//     PlcTask Inputs/GVL_iXlinker.EtherCAT_Master_ATxxxx.Beckhoff_ATH2xxx.Beckhoff_ATH2xxxEK1122.A_0004_ATH2040_0250_0022.InfoData.State <-> InfoData/State
//   PLC/PLC Instance <-> EtherCAT Master ATxxxx/Beckhoff ATH2xxx/Beckhoff ATH2xxxEK1122/A_0005(ATH2040-0250-0023)
//     PlcTask Inputs/GVL_iXlinker.EtherCAT_Master_ATxxxx.Beckhoff_ATH2xxx.Beckhoff_ATH2xxxEK1122.A_0005_ATH2040_0250_0023.CC_Inputs.Status <-> CC Inputs/Status
//     PlcTask Inputs/GVL_iXlinker.EtherCAT_Master_ATxxxx.Beckhoff_ATH2xxx.Beckhoff_ATH2xxxEK1122.A_0005_ATH2040_0250_0023.CC_Inputs.Current_actual_value_Ch[0] <-> CC Inputs/Current actual value Ch.1
//     PlcTask Inputs/GVL_iXlinker.EtherCAT_Master_ATxxxx.Beckhoff_ATH2xxx.Beckhoff_ATH2xxxEK1122.A_0005_ATH2040_0250_0023.CC_Inputs.Current_actual_value_Ch[1] <-> CC Inputs/Current actual value Ch.2
//     PlcTask Inputs/GVL_iXlinker.EtherCAT_Master_ATxxxx.Beckhoff_ATH2xxx.Beckhoff_ATH2xxxEK1122.A_0005_ATH2040_0250_0023.CC_Inputs.Current_actual_value_Ch[2] <-> CC Inputs/Current actual value Ch.3
//     PlcTask Inputs/GVL_iXlinker.EtherCAT_Master_ATxxxx.Beckhoff_ATH2xxx.Beckhoff_ATH2xxxEK1122.A_0005_ATH2040_0250_0023.CC_Inputs.Current_actual_value_Ch[3] <-> CC Inputs/Current actual value Ch.4
//     PlcTask Inputs/GVL_iXlinker.EtherCAT_Master_ATxxxx.Beckhoff_ATH2xxx.Beckhoff_ATH2xxxEK1122.A_0005_ATH2040_0250_0023.CC_Inputs.Current_actual_value_Ch[4] <-> CC Inputs/Current actual value Ch.5
//     PlcTask Inputs/GVL_iXlinker.EtherCAT_Master_ATxxxx.Beckhoff_ATH2xxx.Beckhoff_ATH2xxxEK1122.A_0005_ATH2040_0250_0023.CC_Inputs.Current_actual_value_Ch[5] <-> CC Inputs/Current actual value Ch.6
//     PlcTask Inputs/GVL_iXlinker.EtherCAT_Master_ATxxxx.Beckhoff_ATH2xxx.Beckhoff_ATH2xxxEK1122.A_0005_ATH2040_0250_0023.CC_Inputs.Current_actual_value_Ch[6] <-> CC Inputs/Current actual value Ch.7
//     PlcTask Inputs/GVL_iXlinker.EtherCAT_Master_ATxxxx.Beckhoff_ATH2xxx.Beckhoff_ATH2xxxEK1122.A_0005_ATH2040_0250_0023.CC_Inputs.Current_actual_value_Ch[7] <-> CC Inputs/Current actual value Ch.8
//     PlcTask Inputs/GVL_iXlinker.EtherCAT_Master_ATxxxx.Beckhoff_ATH2xxx.Beckhoff_ATH2xxxEK1122.A_0005_ATH2040_0250_0023.CC_Inputs.Current_actual_value_Ch[8] <-> CC Inputs/Current actual value Ch.9
//     PlcTask Inputs/GVL_iXlinker.EtherCAT_Master_ATxxxx.Beckhoff_ATH2xxx.Beckhoff_ATH2xxxEK1122.A_0005_ATH2040_0250_0023.CC_Inputs.Current_actual_value_Ch[9] <-> CC Inputs/Current actual value Ch.10
//     PlcTask Inputs/GVL_iXlinker.EtherCAT_Master_ATxxxx.Beckhoff_ATH2xxx.Beckhoff_ATH2xxxEK1122.A_0005_ATH2040_0250_0023.CC_Inputs.Current_actual_value_Ch[10] <-> CC Inputs/Current actual value Ch.11
//     PlcTask Inputs/GVL_iXlinker.EtherCAT_Master_ATxxxx.Beckhoff_ATH2xxx.Beckhoff_ATH2xxxEK1122.A_0005_ATH2040_0250_0023.CC_Inputs.Current_actual_value_Ch[11] <-> CC Inputs/Current actual value Ch.12
//     PlcTask Inputs/GVL_iXlinker.EtherCAT_Master_ATxxxx.Beckhoff_ATH2xxx.Beckhoff_ATH2xxxEK1122.A_0005_ATH2040_0250_0023.CC_Inputs.Current_actual_value_Ch[12] <-> CC Inputs/Current actual value Ch.13
//     PlcTask Inputs/GVL_iXlinker.EtherCAT_Master_ATxxxx.Beckhoff_ATH2xxx.Beckhoff_ATH2xxxEK1122.A_0005_ATH2040_0250_0023.CC_Inputs.Current_actual_value_Ch[13] <-> CC Inputs/Current actual value Ch.14
//     PlcTask Inputs/GVL_iXlinker.EtherCAT_Master_ATxxxx.Beckhoff_ATH2xxx.Beckhoff_ATH2xxxEK1122.A_0005_ATH2040_0250_0023.CC_Inputs.Current_actual_value_Ch[14] <-> CC Inputs/Current actual value Ch.15
//     PlcTask Outputs/GVL_iXlinker.EtherCAT_Master_ATxxxx.Beckhoff_ATH2xxx.Beckhoff_ATH2xxxEK1122.A_0005_ATH2040_0250_0023.CC_Outputs.Control <-> CC Outputs/Control
//     PlcTask Outputs/GVL_iXlinker.EtherCAT_Master_ATxxxx.Beckhoff_ATH2xxx.Beckhoff_ATH2xxxEK1122.A_0005_ATH2040_0250_0023.CC_Outputs.Current_setpoint_value_Ch[0] <-> CC Outputs/Current setpoint value Ch.1
//     PlcTask Outputs/GVL_iXlinker.EtherCAT_Master_ATxxxx.Beckhoff_ATH2xxx.Beckhoff_ATH2xxxEK1122.A_0005_ATH2040_0250_0023.CC_Outputs.Current_setpoint_value_Ch[1] <-> CC Outputs/Current setpoint value Ch.2
//     PlcTask Outputs/GVL_iXlinker.EtherCAT_Master_ATxxxx.Beckhoff_ATH2xxx.Beckhoff_ATH2xxxEK1122.A_0005_ATH2040_0250_0023.CC_Outputs.Current_setpoint_value_Ch[2] <-> CC Outputs/Current setpoint value Ch.3
//     PlcTask Outputs/GVL_iXlinker.EtherCAT_Master_ATxxxx.Beckhoff_ATH2xxx.Beckhoff_ATH2xxxEK1122.A_0005_ATH2040_0250_0023.CC_Outputs.Current_setpoint_value_Ch[3] <-> CC Outputs/Current setpoint value Ch.4
//     PlcTask Outputs/GVL_iXlinker.EtherCAT_Master_ATxxxx.Beckhoff_ATH2xxx.Beckhoff_ATH2xxxEK1122.A_0005_ATH2040_0250_0023.CC_Outputs.Current_setpoint_value_Ch[4] <-> CC Outputs/Current setpoint value Ch.5
//     PlcTask Outputs/GVL_iXlinker.EtherCAT_Master_ATxxxx.Beckhoff_ATH2xxx.Beckhoff_ATH2xxxEK1122.A_0005_ATH2040_0250_0023.CC_Outputs.Current_setpoint_value_Ch[5] <-> CC Outputs/Current setpoint value Ch.6
//     PlcTask Outputs/GVL_iXlinker.EtherCAT_Master_ATxxxx.Beckhoff_ATH2xxx.Beckhoff_ATH2xxxEK1122.A_0005_ATH2040_0250_0023.CC_Outputs.Current_setpoint_value_Ch[6] <-> CC Outputs/Current setpoint value Ch.7
//     PlcTask Outputs/GVL_iXlinker.EtherCAT_Master_ATxxxx.Beckhoff_ATH2xxx.Beckhoff_ATH2xxxEK1122.A_0005_ATH2040_0250_0023.CC_Outputs.Current_setpoint_value_Ch[7] <-> CC Outputs/Current setpoint value Ch.8
//     PlcTask Outputs/GVL_iXlinker.EtherCAT_Master_ATxxxx.Beckhoff_ATH2xxx.Beckhoff_ATH2xxxEK1122.A_0005_ATH2040_0250_0023.CC_Outputs.Current_setpoint_value_Ch[8] <-> CC Outputs/Current setpoint value Ch.9
//     PlcTask Outputs/GVL_iXlinker.EtherCAT_Master_ATxxxx.Beckhoff_ATH2xxx.Beckhoff_ATH2xxxEK1122.A_0005_ATH2040_0250_0023.CC_Outputs.Current_setpoint_value_Ch[9] <-> CC Outputs/Current setpoint value Ch.10
//     PlcTask Outputs/GVL_iXlinker.EtherCAT_Master_ATxxxx.Beckhoff_ATH2xxx.Beckhoff_ATH2xxxEK1122.A_0005_ATH2040_0250_0023.CC_Outputs.Current_setpoint_value_Ch[10] <-> CC Outputs/Current setpoint value Ch.11
//     PlcTask Outputs/GVL_iXlinker.EtherCAT_Master_ATxxxx.Beckhoff_ATH2xxx.Beckhoff_ATH2xxxEK1122.A_0005_ATH2040_0250_0023.CC_Outputs.Current_setpoint_value_Ch[11] <-> CC Outputs/Current setpoint value Ch.12
//     PlcTask Outputs/GVL_iXlinker.EtherCAT_Master_ATxxxx.Beckhoff_ATH2xxx.Beckhoff_ATH2xxxEK1122.A_0005_ATH2040_0250_0023.CC_Outputs.Current_setpoint_value_Ch[12] <-> CC Outputs/Current setpoint value Ch.13
//     PlcTask Outputs/GVL_iXlinker.EtherCAT_Master_ATxxxx.Beckhoff_ATH2xxx.Beckhoff_ATH2xxxEK1122.A_0005_ATH2040_0250_0023.CC_Outputs.Current_setpoint_value_Ch[13] <-> CC Outputs/Current setpoint value Ch.14
//     PlcTask Outputs/GVL_iXlinker.EtherCAT_Master_ATxxxx.Beckhoff_ATH2xxx.Beckhoff_ATH2xxxEK1122.A_0005_ATH2040_0250_0023.CC_Outputs.Current_setpoint_value_Ch[14] <-> CC Outputs/Current setpoint value Ch.15
//     PlcTask Inputs/GVL_iXlinker.EtherCAT_Master_ATxxxx.Beckhoff_ATH2xxx.Beckhoff_ATH2xxxEK1122.A_0005_ATH2040_0250_0023.WcState.WcState <-> WcState/WcState
//     PlcTask Inputs/GVL_iXlinker.EtherCAT_Master_ATxxxx.Beckhoff_ATH2xxx.Beckhoff_ATH2xxxEK1122.A_0005_ATH2040_0250_0023.WcState.InputToggle <-> WcState/InputToggle
//     PlcTask Inputs/GVL_iXlinker.EtherCAT_Master_ATxxxx.Beckhoff_ATH2xxx.Beckhoff_ATH2xxxEK1122.A_0005_ATH2040_0250_0023.InfoData.AdsAddr <-> InfoData/AdsAddr
//     PlcTask Inputs/GVL_iXlinker.EtherCAT_Master_ATxxxx.Beckhoff_ATH2xxx.Beckhoff_ATH2xxxEK1122.A_0005_ATH2040_0250_0023.InfoData.DcOutputShift <-> InfoData/DcOutputShift
//     PlcTask Inputs/GVL_iXlinker.EtherCAT_Master_ATxxxx.Beckhoff_ATH2xxx.Beckhoff_ATH2xxxEK1122.A_0005_ATH2040_0250_0023.InfoData.DcInputShift <-> InfoData/DcInputShift
//     PlcTask Inputs/GVL_iXlinker.EtherCAT_Master_ATxxxx.Beckhoff_ATH2xxx.Beckhoff_ATH2xxxEK1122.A_0005_ATH2040_0250_0023.InfoData.State <-> InfoData/State
//   PLC/PLC Instance <-> EtherCAT Master ATxxxx/Beckhoff ATH2xxx/Beckhoff ATH2xxxEK1122/A_0006(ATH2040-0250-0024)
//     PlcTask Inputs/GVL_iXlinker.EtherCAT_Master_ATxxxx.Beckhoff_ATH2xxx.Beckhoff_ATH2xxxEK1122.A_0006_ATH2040_0250_0024.CC_Inputs.Status <-> CC Inputs/Status
//     PlcTask Inputs/GVL_iXlinker.EtherCAT_Master_ATxxxx.Beckhoff_ATH2xxx.Beckhoff_ATH2xxxEK1122.A_0006_ATH2040_0250_0024.CC_Inputs.Current_actual_value_Ch[0] <-> CC Inputs/Current actual value Ch.1
//     PlcTask Inputs/GVL_iXlinker.EtherCAT_Master_ATxxxx.Beckhoff_ATH2xxx.Beckhoff_ATH2xxxEK1122.A_0006_ATH2040_0250_0024.CC_Inputs.Current_actual_value_Ch[1] <-> CC Inputs/Current actual value Ch.2
//     PlcTask Inputs/GVL_iXlinker.EtherCAT_Master_ATxxxx.Beckhoff_ATH2xxx.Beckhoff_ATH2xxxEK1122.A_0006_ATH2040_0250_0024.CC_Inputs.Current_actual_value_Ch[2] <-> CC Inputs/Current actual value Ch.3
//     PlcTask Inputs/GVL_iXlinker.EtherCAT_Master_ATxxxx.Beckhoff_ATH2xxx.Beckhoff_ATH2xxxEK1122.A_0006_ATH2040_0250_0024.CC_Inputs.Current_actual_value_Ch[3] <-> CC Inputs/Current actual value Ch.4
//     PlcTask Inputs/GVL_iXlinker.EtherCAT_Master_ATxxxx.Beckhoff_ATH2xxx.Beckhoff_ATH2xxxEK1122.A_0006_ATH2040_0250_0024.CC_Inputs.Current_actual_value_Ch[4] <-> CC Inputs/Current actual value Ch.5
//     PlcTask Inputs/GVL_iXlinker.EtherCAT_Master_ATxxxx.Beckhoff_ATH2xxx.Beckhoff_ATH2xxxEK1122.A_0006_ATH2040_0250_0024.CC_Inputs.Current_actual_value_Ch[5] <-> CC Inputs/Current actual value Ch.6
//     PlcTask Inputs/GVL_iXlinker.EtherCAT_Master_ATxxxx.Beckhoff_ATH2xxx.Beckhoff_ATH2xxxEK1122.A_0006_ATH2040_0250_0024.CC_Inputs.Current_actual_value_Ch[6] <-> CC Inputs/Current actual value Ch.7
//     PlcTask Inputs/GVL_iXlinker.EtherCAT_Master_ATxxxx.Beckhoff_ATH2xxx.Beckhoff_ATH2xxxEK1122.A_0006_ATH2040_0250_0024.CC_Inputs.Current_actual_value_Ch[7] <-> CC Inputs/Current actual value Ch.8
//     PlcTask Inputs/GVL_iXlinker.EtherCAT_Master_ATxxxx.Beckhoff_ATH2xxx.Beckhoff_ATH2xxxEK1122.A_0006_ATH2040_0250_0024.CC_Inputs.Current_actual_value_Ch[8] <-> CC Inputs/Current actual value Ch.9
//     PlcTask Inputs/GVL_iXlinker.EtherCAT_Master_ATxxxx.Beckhoff_ATH2xxx.Beckhoff_ATH2xxxEK1122.A_0006_ATH2040_0250_0024.CC_Inputs.Current_actual_value_Ch[9] <-> CC Inputs/Current actual value Ch.10
//     PlcTask Inputs/GVL_iXlinker.EtherCAT_Master_ATxxxx.Beckhoff_ATH2xxx.Beckhoff_ATH2xxxEK1122.A_0006_ATH2040_0250_0024.CC_Inputs.Current_actual_value_Ch[10] <-> CC Inputs/Current actual value Ch.11
//     PlcTask Inputs/GVL_iXlinker.EtherCAT_Master_ATxxxx.Beckhoff_ATH2xxx.Beckhoff_ATH2xxxEK1122.A_0006_ATH2040_0250_0024.CC_Inputs.Current_actual_value_Ch[11] <-> CC Inputs/Current actual value Ch.12
//     PlcTask Inputs/GVL_iXlinker.EtherCAT_Master_ATxxxx.Beckhoff_ATH2xxx.Beckhoff_ATH2xxxEK1122.A_0006_ATH2040_0250_0024.CC_Inputs.Current_actual_value_Ch[12] <-> CC Inputs/Current actual value Ch.13
//     PlcTask Inputs/GVL_iXlinker.EtherCAT_Master_ATxxxx.Beckhoff_ATH2xxx.Beckhoff_ATH2xxxEK1122.A_0006_ATH2040_0250_0024.CC_Inputs.Current_actual_value_Ch[13] <-> CC Inputs/Current actual value Ch.14
//     PlcTask Inputs/GVL_iXlinker.EtherCAT_Master_ATxxxx.Beckhoff_ATH2xxx.Beckhoff_ATH2xxxEK1122.A_0006_ATH2040_0250_0024.CC_Inputs.Current_actual_value_Ch[14] <-> CC Inputs/Current actual value Ch.15
//     PlcTask Outputs/GVL_iXlinker.EtherCAT_Master_ATxxxx.Beckhoff_ATH2xxx.Beckhoff_ATH2xxxEK1122.A_0006_ATH2040_0250_0024.CC_Outputs.Control <-> CC Outputs/Control
//     PlcTask Outputs/GVL_iXlinker.EtherCAT_Master_ATxxxx.Beckhoff_ATH2xxx.Beckhoff_ATH2xxxEK1122.A_0006_ATH2040_0250_0024.CC_Outputs.Current_setpoint_value_Ch[0] <-> CC Outputs/Current setpoint value Ch.1
//     PlcTask Outputs/GVL_iXlinker.EtherCAT_Master_ATxxxx.Beckhoff_ATH2xxx.Beckhoff_ATH2xxxEK1122.A_0006_ATH2040_0250_0024.CC_Outputs.Current_setpoint_value_Ch[1] <-> CC Outputs/Current setpoint value Ch.2
//     PlcTask Outputs/GVL_iXlinker.EtherCAT_Master_ATxxxx.Beckhoff_ATH2xxx.Beckhoff_ATH2xxxEK1122.A_0006_ATH2040_0250_0024.CC_Outputs.Current_setpoint_value_Ch[2] <-> CC Outputs/Current setpoint value Ch.3
//     PlcTask Outputs/GVL_iXlinker.EtherCAT_Master_ATxxxx.Beckhoff_ATH2xxx.Beckhoff_ATH2xxxEK1122.A_0006_ATH2040_0250_0024.CC_Outputs.Current_setpoint_value_Ch[3] <-> CC Outputs/Current setpoint value Ch.4
//     PlcTask Outputs/GVL_iXlinker.EtherCAT_Master_ATxxxx.Beckhoff_ATH2xxx.Beckhoff_ATH2xxxEK1122.A_0006_ATH2040_0250_0024.CC_Outputs.Current_setpoint_value_Ch[4] <-> CC Outputs/Current setpoint value Ch.5
//     PlcTask Outputs/GVL_iXlinker.EtherCAT_Master_ATxxxx.Beckhoff_ATH2xxx.Beckhoff_ATH2xxxEK1122.A_0006_ATH2040_0250_0024.CC_Outputs.Current_setpoint_value_Ch[5] <-> CC Outputs/Current setpoint value Ch.6
//     PlcTask Outputs/GVL_iXlinker.EtherCAT_Master_ATxxxx.Beckhoff_ATH2xxx.Beckhoff_ATH2xxxEK1122.A_0006_ATH2040_0250_0024.CC_Outputs.Current_setpoint_value_Ch[6] <-> CC Outputs/Current setpoint value Ch.7
//     PlcTask Outputs/GVL_iXlinker.EtherCAT_Master_ATxxxx.Beckhoff_ATH2xxx.Beckhoff_ATH2xxxEK1122.A_0006_ATH2040_0250_0024.CC_Outputs.Current_setpoint_value_Ch[7] <-> CC Outputs/Current setpoint value Ch.8
//     PlcTask Outputs/GVL_iXlinker.EtherCAT_Master_ATxxxx.Beckhoff_ATH2xxx.Beckhoff_ATH2xxxEK1122.A_0006_ATH2040_0250_0024.CC_Outputs.Current_setpoint_value_Ch[8] <-> CC Outputs/Current setpoint value Ch.9
//     PlcTask Outputs/GVL_iXlinker.EtherCAT_Master_ATxxxx.Beckhoff_ATH2xxx.Beckhoff_ATH2xxxEK1122.A_0006_ATH2040_0250_0024.CC_Outputs.Current_setpoint_value_Ch[9] <-> CC Outputs/Current setpoint value Ch.10
//     PlcTask Outputs/GVL_iXlinker.EtherCAT_Master_ATxxxx.Beckhoff_ATH2xxx.Beckhoff_ATH2xxxEK1122.A_0006_ATH2040_0250_0024.CC_Outputs.Current_setpoint_value_Ch[10] <-> CC Outputs/Current setpoint value Ch.11
//     PlcTask Outputs/GVL_iXlinker.EtherCAT_Master_ATxxxx.Beckhoff_ATH2xxx.Beckhoff_ATH2xxxEK1122.A_0006_ATH2040_0250_0024.CC_Outputs.Current_setpoint_value_Ch[11] <-> CC Outputs/Current setpoint value Ch.12
//     PlcTask Outputs/GVL_iXlinker.EtherCAT_Master_ATxxxx.Beckhoff_ATH2xxx.Beckhoff_ATH2xxxEK1122.A_0006_ATH2040_0250_0024.CC_Outputs.Current_setpoint_value_Ch[12] <-> CC Outputs/Current setpoint value Ch.13
//     PlcTask Outputs/GVL_iXlinker.EtherCAT_Master_ATxxxx.Beckhoff_ATH2xxx.Beckhoff_ATH2xxxEK1122.A_0006_ATH2040_0250_0024.CC_Outputs.Current_setpoint_value_Ch[13] <-> CC Outputs/Current setpoint value Ch.14
//     PlcTask Outputs/GVL_iXlinker.EtherCAT_Master_ATxxxx.Beckhoff_ATH2xxx.Beckhoff_ATH2xxxEK1122.A_0006_ATH2040_0250_0024.CC_Outputs.Current_setpoint_value_Ch[14] <-> CC Outputs/Current setpoint value Ch.15
//     PlcTask Inputs/GVL_iXlinker.EtherCAT_Master_ATxxxx.Beckhoff_ATH2xxx.Beckhoff_ATH2xxxEK1122.A_0006_ATH2040_0250_0024.WcState.WcState <-> WcState/WcState
//     PlcTask Inputs/GVL_iXlinker.EtherCAT_Master_ATxxxx.Beckhoff_ATH2xxx.Beckhoff_ATH2xxxEK1122.A_0006_ATH2040_0250_0024.WcState.InputToggle <-> WcState/InputToggle
//     PlcTask Inputs/GVL_iXlinker.EtherCAT_Master_ATxxxx.Beckhoff_ATH2xxx.Beckhoff_ATH2xxxEK1122.A_0006_ATH2040_0250_0024.InfoData.AdsAddr <-> InfoData/AdsAddr
//     PlcTask Inputs/GVL_iXlinker.EtherCAT_Master_ATxxxx.Beckhoff_ATH2xxx.Beckhoff_ATH2xxxEK1122.A_0006_ATH2040_0250_0024.InfoData.DcOutputShift <-> InfoData/DcOutputShift
//     PlcTask Inputs/GVL_iXlinker.EtherCAT_Master_ATxxxx.Beckhoff_ATH2xxx.Beckhoff_ATH2xxxEK1122.A_0006_ATH2040_0250_0024.InfoData.DcInputShift <-> InfoData/DcInputShift
//     PlcTask Inputs/GVL_iXlinker.EtherCAT_Master_ATxxxx.Beckhoff_ATH2xxx.Beckhoff_ATH2xxxEK1122.A_0006_ATH2040_0250_0024.InfoData.State <-> InfoData/State
//   PLC/PLC Instance <-> EtherCAT Master ATxxxx/Beckhoff ATH2xxx/Beckhoff ATH2xxxEK1122/A_0007(ATH2050-0500-0022)
//     PlcTask Inputs/GVL_iXlinker.EtherCAT_Master_ATxxxx.Beckhoff_ATH2xxx.Beckhoff_ATH2xxxEK1122.A_0007_ATH2050_0500_0022.CC_Inputs.Status <-> CC Inputs/Status
//     PlcTask Inputs/GVL_iXlinker.EtherCAT_Master_ATxxxx.Beckhoff_ATH2xxx.Beckhoff_ATH2xxxEK1122.A_0007_ATH2050_0500_0022.CC_Inputs.Current_actual_value_Ch[0] <-> CC Inputs/Current actual value Ch.1
//     PlcTask Inputs/GVL_iXlinker.EtherCAT_Master_ATxxxx.Beckhoff_ATH2xxx.Beckhoff_ATH2xxxEK1122.A_0007_ATH2050_0500_0022.CC_Inputs.Current_actual_value_Ch[1] <-> CC Inputs/Current actual value Ch.2
//     PlcTask Inputs/GVL_iXlinker.EtherCAT_Master_ATxxxx.Beckhoff_ATH2xxx.Beckhoff_ATH2xxxEK1122.A_0007_ATH2050_0500_0022.CC_Inputs.Current_actual_value_Ch[2] <-> CC Inputs/Current actual value Ch.3
//     PlcTask Inputs/GVL_iXlinker.EtherCAT_Master_ATxxxx.Beckhoff_ATH2xxx.Beckhoff_ATH2xxxEK1122.A_0007_ATH2050_0500_0022.CC_Inputs.Current_actual_value_Ch[3] <-> CC Inputs/Current actual value Ch.4
//     PlcTask Inputs/GVL_iXlinker.EtherCAT_Master_ATxxxx.Beckhoff_ATH2xxx.Beckhoff_ATH2xxxEK1122.A_0007_ATH2050_0500_0022.CC_Inputs.Current_actual_value_Ch[4] <-> CC Inputs/Current actual value Ch.5
//     PlcTask Inputs/GVL_iXlinker.EtherCAT_Master_ATxxxx.Beckhoff_ATH2xxx.Beckhoff_ATH2xxxEK1122.A_0007_ATH2050_0500_0022.CC_Inputs.Current_actual_value_Ch[5] <-> CC Inputs/Current actual value Ch.6
//     PlcTask Inputs/GVL_iXlinker.EtherCAT_Master_ATxxxx.Beckhoff_ATH2xxx.Beckhoff_ATH2xxxEK1122.A_0007_ATH2050_0500_0022.CC_Inputs.Current_actual_value_Ch[6] <-> CC Inputs/Current actual value Ch.7
//     PlcTask Inputs/GVL_iXlinker.EtherCAT_Master_ATxxxx.Beckhoff_ATH2xxx.Beckhoff_ATH2xxxEK1122.A_0007_ATH2050_0500_0022.CC_Inputs.Current_actual_value_Ch[7] <-> CC Inputs/Current actual value Ch.8
//     PlcTask Inputs/GVL_iXlinker.EtherCAT_Master_ATxxxx.Beckhoff_ATH2xxx.Beckhoff_ATH2xxxEK1122.A_0007_ATH2050_0500_0022.CC_Inputs.Current_actual_value_Ch[8] <-> CC Inputs/Current actual value Ch.9
//     PlcTask Inputs/GVL_iXlinker.EtherCAT_Master_ATxxxx.Beckhoff_ATH2xxx.Beckhoff_ATH2xxxEK1122.A_0007_ATH2050_0500_0022.CC_Inputs.Current_actual_value_Ch[9] <-> CC Inputs/Current actual value Ch.10
//     PlcTask Inputs/GVL_iXlinker.EtherCAT_Master_ATxxxx.Beckhoff_ATH2xxx.Beckhoff_ATH2xxxEK1122.A_0007_ATH2050_0500_0022.CC_Inputs.Current_actual_value_Ch[10] <-> CC Inputs/Current actual value Ch.11
//     PlcTask Inputs/GVL_iXlinker.EtherCAT_Master_ATxxxx.Beckhoff_ATH2xxx.Beckhoff_ATH2xxxEK1122.A_0007_ATH2050_0500_0022.CC_Inputs.Current_actual_value_Ch[11] <-> CC Inputs/Current actual value Ch.12
//     PlcTask Inputs/GVL_iXlinker.EtherCAT_Master_ATxxxx.Beckhoff_ATH2xxx.Beckhoff_ATH2xxxEK1122.A_0007_ATH2050_0500_0022.CC_Inputs.Current_actual_value_Ch[12] <-> CC Inputs/Current actual value Ch.13
//     PlcTask Inputs/GVL_iXlinker.EtherCAT_Master_ATxxxx.Beckhoff_ATH2xxx.Beckhoff_ATH2xxxEK1122.A_0007_ATH2050_0500_0022.CC_Inputs.Current_actual_value_Ch[13] <-> CC Inputs/Current actual value Ch.14
//     PlcTask Inputs/GVL_iXlinker.EtherCAT_Master_ATxxxx.Beckhoff_ATH2xxx.Beckhoff_ATH2xxxEK1122.A_0007_ATH2050_0500_0022.CC_Inputs.Current_actual_value_Ch[14] <-> CC Inputs/Current actual value Ch.15
//     PlcTask Outputs/GVL_iXlinker.EtherCAT_Master_ATxxxx.Beckhoff_ATH2xxx.Beckhoff_ATH2xxxEK1122.A_0007_ATH2050_0500_0022.CC_Outputs.Control <-> CC Outputs/Control
//     PlcTask Outputs/GVL_iXlinker.EtherCAT_Master_ATxxxx.Beckhoff_ATH2xxx.Beckhoff_ATH2xxxEK1122.A_0007_ATH2050_0500_0022.CC_Outputs.Current_setpoint_value_Ch[0] <-> CC Outputs/Current setpoint value Ch.1
//     PlcTask Outputs/GVL_iXlinker.EtherCAT_Master_ATxxxx.Beckhoff_ATH2xxx.Beckhoff_ATH2xxxEK1122.A_0007_ATH2050_0500_0022.CC_Outputs.Current_setpoint_value_Ch[1] <-> CC Outputs/Current setpoint value Ch.2
//     PlcTask Outputs/GVL_iXlinker.EtherCAT_Master_ATxxxx.Beckhoff_ATH2xxx.Beckhoff_ATH2xxxEK1122.A_0007_ATH2050_0500_0022.CC_Outputs.Current_setpoint_value_Ch[2] <-> CC Outputs/Current setpoint value Ch.3
//     PlcTask Outputs/GVL_iXlinker.EtherCAT_Master_ATxxxx.Beckhoff_ATH2xxx.Beckhoff_ATH2xxxEK1122.A_0007_ATH2050_0500_0022.CC_Outputs.Current_setpoint_value_Ch[3] <-> CC Outputs/Current setpoint value Ch.4
//     PlcTask Outputs/GVL_iXlinker.EtherCAT_Master_ATxxxx.Beckhoff_ATH2xxx.Beckhoff_ATH2xxxEK1122.A_0007_ATH2050_0500_0022.CC_Outputs.Current_setpoint_value_Ch[4] <-> CC Outputs/Current setpoint value Ch.5
//     PlcTask Outputs/GVL_iXlinker.EtherCAT_Master_ATxxxx.Beckhoff_ATH2xxx.Beckhoff_ATH2xxxEK1122.A_0007_ATH2050_0500_0022.CC_Outputs.Current_setpoint_value_Ch[5] <-> CC Outputs/Current setpoint value Ch.6
//     PlcTask Outputs/GVL_iXlinker.EtherCAT_Master_ATxxxx.Beckhoff_ATH2xxx.Beckhoff_ATH2xxxEK1122.A_0007_ATH2050_0500_0022.CC_Outputs.Current_setpoint_value_Ch[6] <-> CC Outputs/Current setpoint value Ch.7
//     PlcTask Outputs/GVL_iXlinker.EtherCAT_Master_ATxxxx.Beckhoff_ATH2xxx.Beckhoff_ATH2xxxEK1122.A_0007_ATH2050_0500_0022.CC_Outputs.Current_setpoint_value_Ch[7] <-> CC Outputs/Current setpoint value Ch.8
//     PlcTask Outputs/GVL_iXlinker.EtherCAT_Master_ATxxxx.Beckhoff_ATH2xxx.Beckhoff_ATH2xxxEK1122.A_0007_ATH2050_0500_0022.CC_Outputs.Current_setpoint_value_Ch[8] <-> CC Outputs/Current setpoint value Ch.9
//     PlcTask Outputs/GVL_iXlinker.EtherCAT_Master_ATxxxx.Beckhoff_ATH2xxx.Beckhoff_ATH2xxxEK1122.A_0007_ATH2050_0500_0022.CC_Outputs.Current_setpoint_value_Ch[9] <-> CC Outputs/Current setpoint value Ch.10
//     PlcTask Outputs/GVL_iXlinker.EtherCAT_Master_ATxxxx.Beckhoff_ATH2xxx.Beckhoff_ATH2xxxEK1122.A_0007_ATH2050_0500_0022.CC_Outputs.Current_setpoint_value_Ch[10] <-> CC Outputs/Current setpoint value Ch.11
//     PlcTask Outputs/GVL_iXlinker.EtherCAT_Master_ATxxxx.Beckhoff_ATH2xxx.Beckhoff_ATH2xxxEK1122.A_0007_ATH2050_0500_0022.CC_Outputs.Current_setpoint_value_Ch[11] <-> CC Outputs/Current setpoint value Ch.12
//     PlcTask Outputs/GVL_iXlinker.EtherCAT_Master_ATxxxx.Beckhoff_ATH2xxx.Beckhoff_ATH2xxxEK1122.A_0007_ATH2050_0500_0022.CC_Outputs.Current_setpoint_value_Ch[12] <-> CC Outputs/Current setpoint value Ch.13
//     PlcTask Outputs/GVL_iXlinker.EtherCAT_Master_ATxxxx.Beckhoff_ATH2xxx.Beckhoff_ATH2xxxEK1122.A_0007_ATH2050_0500_0022.CC_Outputs.Current_setpoint_value_Ch[13] <-> CC Outputs/Current setpoint value Ch.14
//     PlcTask Outputs/GVL_iXlinker.EtherCAT_Master_ATxxxx.Beckhoff_ATH2xxx.Beckhoff_ATH2xxxEK1122.A_0007_ATH2050_0500_0022.CC_Outputs.Current_setpoint_value_Ch[14] <-> CC Outputs/Current setpoint value Ch.15
//     PlcTask Inputs/GVL_iXlinker.EtherCAT_Master_ATxxxx.Beckhoff_ATH2xxx.Beckhoff_ATH2xxxEK1122.A_0007_ATH2050_0500_0022.WcState.WcState <-> WcState/WcState
//     PlcTask Inputs/GVL_iXlinker.EtherCAT_Master_ATxxxx.Beckhoff_ATH2xxx.Beckhoff_ATH2xxxEK1122.A_0007_ATH2050_0500_0022.WcState.InputToggle <-> WcState/InputToggle
//     PlcTask Inputs/GVL_iXlinker.EtherCAT_Master_ATxxxx.Beckhoff_ATH2xxx.Beckhoff_ATH2xxxEK1122.A_0007_ATH2050_0500_0022.InfoData.AdsAddr <-> InfoData/AdsAddr
//     PlcTask Inputs/GVL_iXlinker.EtherCAT_Master_ATxxxx.Beckhoff_ATH2xxx.Beckhoff_ATH2xxxEK1122.A_0007_ATH2050_0500_0022.InfoData.DcOutputShift <-> InfoData/DcOutputShift
//     PlcTask Inputs/GVL_iXlinker.EtherCAT_Master_ATxxxx.Beckhoff_ATH2xxx.Beckhoff_ATH2xxxEK1122.A_0007_ATH2050_0500_0022.InfoData.DcInputShift <-> InfoData/DcInputShift
//     PlcTask Inputs/GVL_iXlinker.EtherCAT_Master_ATxxxx.Beckhoff_ATH2xxx.Beckhoff_ATH2xxxEK1122.A_0007_ATH2050_0500_0022.InfoData.State <-> InfoData/State
//   PLC/PLC Instance <-> EtherCAT Master ATxxxx/Beckhoff ATH2xxx/Beckhoff ATH2xxxEK1122/A_0008(ATH2050-0500-0023)
//     PlcTask Inputs/GVL_iXlinker.EtherCAT_Master_ATxxxx.Beckhoff_ATH2xxx.Beckhoff_ATH2xxxEK1122.A_0008_ATH2050_0500_0023.CC_Inputs.Status <-> CC Inputs/Status
//     PlcTask Inputs/GVL_iXlinker.EtherCAT_Master_ATxxxx.Beckhoff_ATH2xxx.Beckhoff_ATH2xxxEK1122.A_0008_ATH2050_0500_0023.CC_Inputs.Current_actual_value_Ch[0] <-> CC Inputs/Current actual value Ch.1
//     PlcTask Inputs/GVL_iXlinker.EtherCAT_Master_ATxxxx.Beckhoff_ATH2xxx.Beckhoff_ATH2xxxEK1122.A_0008_ATH2050_0500_0023.CC_Inputs.Current_actual_value_Ch[1] <-> CC Inputs/Current actual value Ch.2
//     PlcTask Inputs/GVL_iXlinker.EtherCAT_Master_ATxxxx.Beckhoff_ATH2xxx.Beckhoff_ATH2xxxEK1122.A_0008_ATH2050_0500_0023.CC_Inputs.Current_actual_value_Ch[2] <-> CC Inputs/Current actual value Ch.3
//     PlcTask Inputs/GVL_iXlinker.EtherCAT_Master_ATxxxx.Beckhoff_ATH2xxx.Beckhoff_ATH2xxxEK1122.A_0008_ATH2050_0500_0023.CC_Inputs.Current_actual_value_Ch[3] <-> CC Inputs/Current actual value Ch.4
//     PlcTask Inputs/GVL_iXlinker.EtherCAT_Master_ATxxxx.Beckhoff_ATH2xxx.Beckhoff_ATH2xxxEK1122.A_0008_ATH2050_0500_0023.CC_Inputs.Current_actual_value_Ch[4] <-> CC Inputs/Current actual value Ch.5
//     PlcTask Inputs/GVL_iXlinker.EtherCAT_Master_ATxxxx.Beckhoff_ATH2xxx.Beckhoff_ATH2xxxEK1122.A_0008_ATH2050_0500_0023.CC_Inputs.Current_actual_value_Ch[5] <-> CC Inputs/Current actual value Ch.6
//     PlcTask Inputs/GVL_iXlinker.EtherCAT_Master_ATxxxx.Beckhoff_ATH2xxx.Beckhoff_ATH2xxxEK1122.A_0008_ATH2050_0500_0023.CC_Inputs.Current_actual_value_Ch[6] <-> CC Inputs/Current actual value Ch.7
//     PlcTask Inputs/GVL_iXlinker.EtherCAT_Master_ATxxxx.Beckhoff_ATH2xxx.Beckhoff_ATH2xxxEK1122.A_0008_ATH2050_0500_0023.CC_Inputs.Current_actual_value_Ch[7] <-> CC Inputs/Current actual value Ch.8
//     PlcTask Inputs/GVL_iXlinker.EtherCAT_Master_ATxxxx.Beckhoff_ATH2xxx.Beckhoff_ATH2xxxEK1122.A_0008_ATH2050_0500_0023.CC_Inputs.Current_actual_value_Ch[8] <-> CC Inputs/Current actual value Ch.9
//     PlcTask Inputs/GVL_iXlinker.EtherCAT_Master_ATxxxx.Beckhoff_ATH2xxx.Beckhoff_ATH2xxxEK1122.A_0008_ATH2050_0500_0023.CC_Inputs.Current_actual_value_Ch[9] <-> CC Inputs/Current actual value Ch.10
//     PlcTask Inputs/GVL_iXlinker.EtherCAT_Master_ATxxxx.Beckhoff_ATH2xxx.Beckhoff_ATH2xxxEK1122.A_0008_ATH2050_0500_0023.CC_Inputs.Current_actual_value_Ch[10] <-> CC Inputs/Current actual value Ch.11
//     PlcTask Inputs/GVL_iXlinker.EtherCAT_Master_ATxxxx.Beckhoff_ATH2xxx.Beckhoff_ATH2xxxEK1122.A_0008_ATH2050_0500_0023.CC_Inputs.Current_actual_value_Ch[11] <-> CC Inputs/Current actual value Ch.12
//     PlcTask Inputs/GVL_iXlinker.EtherCAT_Master_ATxxxx.Beckhoff_ATH2xxx.Beckhoff_ATH2xxxEK1122.A_0008_ATH2050_0500_0023.CC_Inputs.Current_actual_value_Ch[12] <-> CC Inputs/Current actual value Ch.13
//     PlcTask Inputs/GVL_iXlinker.EtherCAT_Master_ATxxxx.Beckhoff_ATH2xxx.Beckhoff_ATH2xxxEK1122.A_0008_ATH2050_0500_0023.CC_Inputs.Current_actual_value_Ch[13] <-> CC Inputs/Current actual value Ch.14
//     PlcTask Inputs/GVL_iXlinker.EtherCAT_Master_ATxxxx.Beckhoff_ATH2xxx.Beckhoff_ATH2xxxEK1122.A_0008_ATH2050_0500_0023.CC_Inputs.Current_actual_value_Ch[14] <-> CC Inputs/Current actual value Ch.15
//     PlcTask Outputs/GVL_iXlinker.EtherCAT_Master_ATxxxx.Beckhoff_ATH2xxx.Beckhoff_ATH2xxxEK1122.A_0008_ATH2050_0500_0023.CC_Outputs.Control <-> CC Outputs/Control
//     PlcTask Outputs/GVL_iXlinker.EtherCAT_Master_ATxxxx.Beckhoff_ATH2xxx.Beckhoff_ATH2xxxEK1122.A_0008_ATH2050_0500_0023.CC_Outputs.Current_setpoint_value_Ch[0] <-> CC Outputs/Current setpoint value Ch.1
//     PlcTask Outputs/GVL_iXlinker.EtherCAT_Master_ATxxxx.Beckhoff_ATH2xxx.Beckhoff_ATH2xxxEK1122.A_0008_ATH2050_0500_0023.CC_Outputs.Current_setpoint_value_Ch[1] <-> CC Outputs/Current setpoint value Ch.2
//     PlcTask Outputs/GVL_iXlinker.EtherCAT_Master_ATxxxx.Beckhoff_ATH2xxx.Beckhoff_ATH2xxxEK1122.A_0008_ATH2050_0500_0023.CC_Outputs.Current_setpoint_value_Ch[2] <-> CC Outputs/Current setpoint value Ch.3
//     PlcTask Outputs/GVL_iXlinker.EtherCAT_Master_ATxxxx.Beckhoff_ATH2xxx.Beckhoff_ATH2xxxEK1122.A_0008_ATH2050_0500_0023.CC_Outputs.Current_setpoint_value_Ch[3] <-> CC Outputs/Current setpoint value Ch.4
//     PlcTask Outputs/GVL_iXlinker.EtherCAT_Master_ATxxxx.Beckhoff_ATH2xxx.Beckhoff_ATH2xxxEK1122.A_0008_ATH2050_0500_0023.CC_Outputs.Current_setpoint_value_Ch[4] <-> CC Outputs/Current setpoint value Ch.5
//     PlcTask Outputs/GVL_iXlinker.EtherCAT_Master_ATxxxx.Beckhoff_ATH2xxx.Beckhoff_ATH2xxxEK1122.A_0008_ATH2050_0500_0023.CC_Outputs.Current_setpoint_value_Ch[5] <-> CC Outputs/Current setpoint value Ch.6
//     PlcTask Outputs/GVL_iXlinker.EtherCAT_Master_ATxxxx.Beckhoff_ATH2xxx.Beckhoff_ATH2xxxEK1122.A_0008_ATH2050_0500_0023.CC_Outputs.Current_setpoint_value_Ch[6] <-> CC Outputs/Current setpoint value Ch.7
//     PlcTask Outputs/GVL_iXlinker.EtherCAT_Master_ATxxxx.Beckhoff_ATH2xxx.Beckhoff_ATH2xxxEK1122.A_0008_ATH2050_0500_0023.CC_Outputs.Current_setpoint_value_Ch[7] <-> CC Outputs/Current setpoint value Ch.8
//     PlcTask Outputs/GVL_iXlinker.EtherCAT_Master_ATxxxx.Beckhoff_ATH2xxx.Beckhoff_ATH2xxxEK1122.A_0008_ATH2050_0500_0023.CC_Outputs.Current_setpoint_value_Ch[8] <-> CC Outputs/Current setpoint value Ch.9
//     PlcTask Outputs/GVL_iXlinker.EtherCAT_Master_ATxxxx.Beckhoff_ATH2xxx.Beckhoff_ATH2xxxEK1122.A_0008_ATH2050_0500_0023.CC_Outputs.Current_setpoint_value_Ch[9] <-> CC Outputs/Current setpoint value Ch.10
//     PlcTask Outputs/GVL_iXlinker.EtherCAT_Master_ATxxxx.Beckhoff_ATH2xxx.Beckhoff_ATH2xxxEK1122.A_0008_ATH2050_0500_0023.CC_Outputs.Current_setpoint_value_Ch[10] <-> CC Outputs/Current setpoint value Ch.11
//     PlcTask Outputs/GVL_iXlinker.EtherCAT_Master_ATxxxx.Beckhoff_ATH2xxx.Beckhoff_ATH2xxxEK1122.A_0008_ATH2050_0500_0023.CC_Outputs.Current_setpoint_value_Ch[11] <-> CC Outputs/Current setpoint value Ch.12
//     PlcTask Outputs/GVL_iXlinker.EtherCAT_Master_ATxxxx.Beckhoff_ATH2xxx.Beckhoff_ATH2xxxEK1122.A_0008_ATH2050_0500_0023.CC_Outputs.Current_setpoint_value_Ch[12] <-> CC Outputs/Current setpoint value Ch.13
//     PlcTask Outputs/GVL_iXlinker.EtherCAT_Master_ATxxxx.Beckhoff_ATH2xxx.Beckhoff_ATH2xxxEK1122.A_0008_ATH2050_0500_0023.CC_Outputs.Current_setpoint_value_Ch[13] <-> CC Outputs/Current setpoint value Ch.14
//     PlcTask Outputs/GVL_iXlinker.EtherCAT_Master_ATxxxx.Beckhoff_ATH2xxx.Beckhoff_ATH2xxxEK1122.A_0008_ATH2050_0500_0023.CC_Outputs.Current_setpoint_value_Ch[14] <-> CC Outputs/Current setpoint value Ch.15
//     PlcTask Inputs/GVL_iXlinker.EtherCAT_Master_ATxxxx.Beckhoff_ATH2xxx.Beckhoff_ATH2xxxEK1122.A_0008_ATH2050_0500_0023.WcState.WcState <-> WcState/WcState
//     PlcTask Inputs/GVL_iXlinker.EtherCAT_Master_ATxxxx.Beckhoff_ATH2xxx.Beckhoff_ATH2xxxEK1122.A_0008_ATH2050_0500_0023.WcState.InputToggle <-> WcState/InputToggle
//     PlcTask Inputs/GVL_iXlinker.EtherCAT_Master_ATxxxx.Beckhoff_ATH2xxx.Beckhoff_ATH2xxxEK1122.A_0008_ATH2050_0500_0023.InfoData.AdsAddr <-> InfoData/AdsAddr
//     PlcTask Inputs/GVL_iXlinker.EtherCAT_Master_ATxxxx.Beckhoff_ATH2xxx.Beckhoff_ATH2xxxEK1122.A_0008_ATH2050_0500_0023.InfoData.DcOutputShift <-> InfoData/DcOutputShift
//     PlcTask Inputs/GVL_iXlinker.EtherCAT_Master_ATxxxx.Beckhoff_ATH2xxx.Beckhoff_ATH2xxxEK1122.A_0008_ATH2050_0500_0023.InfoData.DcInputShift <-> InfoData/DcInputShift
//     PlcTask Inputs/GVL_iXlinker.EtherCAT_Master_ATxxxx.Beckhoff_ATH2xxx.Beckhoff_ATH2xxxEK1122.A_0008_ATH2050_0500_0023.InfoData.State <-> InfoData/State
//   PLC/PLC Instance <-> EtherCAT Master ATxxxx/Beckhoff ATH2xxx/Beckhoff ATH2xxxEK1122/A_0009(ATH2050-0500-0024)
//     PlcTask Inputs/GVL_iXlinker.EtherCAT_Master_ATxxxx.Beckhoff_ATH2xxx.Beckhoff_ATH2xxxEK1122.A_0009_ATH2050_0500_0024.CC_Inputs.Status <-> CC Inputs/Status
//     PlcTask Inputs/GVL_iXlinker.EtherCAT_Master_ATxxxx.Beckhoff_ATH2xxx.Beckhoff_ATH2xxxEK1122.A_0009_ATH2050_0500_0024.CC_Inputs.Current_actual_value_Ch[0] <-> CC Inputs/Current actual value Ch.1
//     PlcTask Inputs/GVL_iXlinker.EtherCAT_Master_ATxxxx.Beckhoff_ATH2xxx.Beckhoff_ATH2xxxEK1122.A_0009_ATH2050_0500_0024.CC_Inputs.Current_actual_value_Ch[1] <-> CC Inputs/Current actual value Ch.2
//     PlcTask Inputs/GVL_iXlinker.EtherCAT_Master_ATxxxx.Beckhoff_ATH2xxx.Beckhoff_ATH2xxxEK1122.A_0009_ATH2050_0500_0024.CC_Inputs.Current_actual_value_Ch[2] <-> CC Inputs/Current actual value Ch.3
//     PlcTask Inputs/GVL_iXlinker.EtherCAT_Master_ATxxxx.Beckhoff_ATH2xxx.Beckhoff_ATH2xxxEK1122.A_0009_ATH2050_0500_0024.CC_Inputs.Current_actual_value_Ch[3] <-> CC Inputs/Current actual value Ch.4
//     PlcTask Inputs/GVL_iXlinker.EtherCAT_Master_ATxxxx.Beckhoff_ATH2xxx.Beckhoff_ATH2xxxEK1122.A_0009_ATH2050_0500_0024.CC_Inputs.Current_actual_value_Ch[4] <-> CC Inputs/Current actual value Ch.5
//     PlcTask Inputs/GVL_iXlinker.EtherCAT_Master_ATxxxx.Beckhoff_ATH2xxx.Beckhoff_ATH2xxxEK1122.A_0009_ATH2050_0500_0024.CC_Inputs.Current_actual_value_Ch[5] <-> CC Inputs/Current actual value Ch.6
//     PlcTask Inputs/GVL_iXlinker.EtherCAT_Master_ATxxxx.Beckhoff_ATH2xxx.Beckhoff_ATH2xxxEK1122.A_0009_ATH2050_0500_0024.CC_Inputs.Current_actual_value_Ch[6] <-> CC Inputs/Current actual value Ch.7
//     PlcTask Inputs/GVL_iXlinker.EtherCAT_Master_ATxxxx.Beckhoff_ATH2xxx.Beckhoff_ATH2xxxEK1122.A_0009_ATH2050_0500_0024.CC_Inputs.Current_actual_value_Ch[7] <-> CC Inputs/Current actual value Ch.8
//     PlcTask Inputs/GVL_iXlinker.EtherCAT_Master_ATxxxx.Beckhoff_ATH2xxx.Beckhoff_ATH2xxxEK1122.A_0009_ATH2050_0500_0024.CC_Inputs.Current_actual_value_Ch[8] <-> CC Inputs/Current actual value Ch.9
//     PlcTask Inputs/GVL_iXlinker.EtherCAT_Master_ATxxxx.Beckhoff_ATH2xxx.Beckhoff_ATH2xxxEK1122.A_0009_ATH2050_0500_0024.CC_Inputs.Current_actual_value_Ch[9] <-> CC Inputs/Current actual value Ch.10
//     PlcTask Inputs/GVL_iXlinker.EtherCAT_Master_ATxxxx.Beckhoff_ATH2xxx.Beckhoff_ATH2xxxEK1122.A_0009_ATH2050_0500_0024.CC_Inputs.Current_actual_value_Ch[10] <-> CC Inputs/Current actual value Ch.11
//     PlcTask Inputs/GVL_iXlinker.EtherCAT_Master_ATxxxx.Beckhoff_ATH2xxx.Beckhoff_ATH2xxxEK1122.A_0009_ATH2050_0500_0024.CC_Inputs.Current_actual_value_Ch[11] <-> CC Inputs/Current actual value Ch.12
//     PlcTask Inputs/GVL_iXlinker.EtherCAT_Master_ATxxxx.Beckhoff_ATH2xxx.Beckhoff_ATH2xxxEK1122.A_0009_ATH2050_0500_0024.CC_Inputs.Current_actual_value_Ch[12] <-> CC Inputs/Current actual value Ch.13
//     PlcTask Inputs/GVL_iXlinker.EtherCAT_Master_ATxxxx.Beckhoff_ATH2xxx.Beckhoff_ATH2xxxEK1122.A_0009_ATH2050_0500_0024.CC_Inputs.Current_actual_value_Ch[13] <-> CC Inputs/Current actual value Ch.14
//     PlcTask Inputs/GVL_iXlinker.EtherCAT_Master_ATxxxx.Beckhoff_ATH2xxx.Beckhoff_ATH2xxxEK1122.A_0009_ATH2050_0500_0024.CC_Inputs.Current_actual_value_Ch[14] <-> CC Inputs/Current actual value Ch.15
//     PlcTask Outputs/GVL_iXlinker.EtherCAT_Master_ATxxxx.Beckhoff_ATH2xxx.Beckhoff_ATH2xxxEK1122.A_0009_ATH2050_0500_0024.CC_Outputs.Control <-> CC Outputs/Control
//     PlcTask Outputs/GVL_iXlinker.EtherCAT_Master_ATxxxx.Beckhoff_ATH2xxx.Beckhoff_ATH2xxxEK1122.A_0009_ATH2050_0500_0024.CC_Outputs.Current_setpoint_value_Ch[0] <-> CC Outputs/Current setpoint value Ch.1
//     PlcTask Outputs/GVL_iXlinker.EtherCAT_Master_ATxxxx.Beckhoff_ATH2xxx.Beckhoff_ATH2xxxEK1122.A_0009_ATH2050_0500_0024.CC_Outputs.Current_setpoint_value_Ch[1] <-> CC Outputs/Current setpoint value Ch.2
//     PlcTask Outputs/GVL_iXlinker.EtherCAT_Master_ATxxxx.Beckhoff_ATH2xxx.Beckhoff_ATH2xxxEK1122.A_0009_ATH2050_0500_0024.CC_Outputs.Current_setpoint_value_Ch[2] <-> CC Outputs/Current setpoint value Ch.3
//     PlcTask Outputs/GVL_iXlinker.EtherCAT_Master_ATxxxx.Beckhoff_ATH2xxx.Beckhoff_ATH2xxxEK1122.A_0009_ATH2050_0500_0024.CC_Outputs.Current_setpoint_value_Ch[3] <-> CC Outputs/Current setpoint value Ch.4
//     PlcTask Outputs/GVL_iXlinker.EtherCAT_Master_ATxxxx.Beckhoff_ATH2xxx.Beckhoff_ATH2xxxEK1122.A_0009_ATH2050_0500_0024.CC_Outputs.Current_setpoint_value_Ch[4] <-> CC Outputs/Current setpoint value Ch.5
//     PlcTask Outputs/GVL_iXlinker.EtherCAT_Master_ATxxxx.Beckhoff_ATH2xxx.Beckhoff_ATH2xxxEK1122.A_0009_ATH2050_0500_0024.CC_Outputs.Current_setpoint_value_Ch[5] <-> CC Outputs/Current setpoint value Ch.6
//     PlcTask Outputs/GVL_iXlinker.EtherCAT_Master_ATxxxx.Beckhoff_ATH2xxx.Beckhoff_ATH2xxxEK1122.A_0009_ATH2050_0500_0024.CC_Outputs.Current_setpoint_value_Ch[6] <-> CC Outputs/Current setpoint value Ch.7
//     PlcTask Outputs/GVL_iXlinker.EtherCAT_Master_ATxxxx.Beckhoff_ATH2xxx.Beckhoff_ATH2xxxEK1122.A_0009_ATH2050_0500_0024.CC_Outputs.Current_setpoint_value_Ch[7] <-> CC Outputs/Current setpoint value Ch.8
//     PlcTask Outputs/GVL_iXlinker.EtherCAT_Master_ATxxxx.Beckhoff_ATH2xxx.Beckhoff_ATH2xxxEK1122.A_0009_ATH2050_0500_0024.CC_Outputs.Current_setpoint_value_Ch[8] <-> CC Outputs/Current setpoint value Ch.9
//     PlcTask Outputs/GVL_iXlinker.EtherCAT_Master_ATxxxx.Beckhoff_ATH2xxx.Beckhoff_ATH2xxxEK1122.A_0009_ATH2050_0500_0024.CC_Outputs.Current_setpoint_value_Ch[9] <-> CC Outputs/Current setpoint value Ch.10
//     PlcTask Outputs/GVL_iXlinker.EtherCAT_Master_ATxxxx.Beckhoff_ATH2xxx.Beckhoff_ATH2xxxEK1122.A_0009_ATH2050_0500_0024.CC_Outputs.Current_setpoint_value_Ch[10] <-> CC Outputs/Current setpoint value Ch.11
//     PlcTask Outputs/GVL_iXlinker.EtherCAT_Master_ATxxxx.Beckhoff_ATH2xxx.Beckhoff_ATH2xxxEK1122.A_0009_ATH2050_0500_0024.CC_Outputs.Current_setpoint_value_Ch[11] <-> CC Outputs/Current setpoint value Ch.12
//     PlcTask Outputs/GVL_iXlinker.EtherCAT_Master_ATxxxx.Beckhoff_ATH2xxx.Beckhoff_ATH2xxxEK1122.A_0009_ATH2050_0500_0024.CC_Outputs.Current_setpoint_value_Ch[12] <-> CC Outputs/Current setpoint value Ch.13
//     PlcTask Outputs/GVL_iXlinker.EtherCAT_Master_ATxxxx.Beckhoff_ATH2xxx.Beckhoff_ATH2xxxEK1122.A_0009_ATH2050_0500_0024.CC_Outputs.Current_setpoint_value_Ch[13] <-> CC Outputs/Current setpoint value Ch.14
//     PlcTask Outputs/GVL_iXlinker.EtherCAT_Master_ATxxxx.Beckhoff_ATH2xxx.Beckhoff_ATH2xxxEK1122.A_0009_ATH2050_0500_0024.CC_Outputs.Current_setpoint_value_Ch[14] <-> CC Outputs/Current setpoint value Ch.15
//     PlcTask Inputs/GVL_iXlinker.EtherCAT_Master_ATxxxx.Beckhoff_ATH2xxx.Beckhoff_ATH2xxxEK1122.A_0009_ATH2050_0500_0024.WcState.WcState <-> WcState/WcState
//     PlcTask Inputs/GVL_iXlinker.EtherCAT_Master_ATxxxx.Beckhoff_ATH2xxx.Beckhoff_ATH2xxxEK1122.A_0009_ATH2050_0500_0024.WcState.InputToggle <-> WcState/InputToggle
//     PlcTask Inputs/GVL_iXlinker.EtherCAT_Master_ATxxxx.Beckhoff_ATH2xxx.Beckhoff_ATH2xxxEK1122.A_0009_ATH2050_0500_0024.InfoData.AdsAddr <-> InfoData/AdsAddr
//     PlcTask Inputs/GVL_iXlinker.EtherCAT_Master_ATxxxx.Beckhoff_ATH2xxx.Beckhoff_ATH2xxxEK1122.A_0009_ATH2050_0500_0024.InfoData.DcOutputShift <-> InfoData/DcOutputShift
//     PlcTask Inputs/GVL_iXlinker.EtherCAT_Master_ATxxxx.Beckhoff_ATH2xxx.Beckhoff_ATH2xxxEK1122.A_0009_ATH2050_0500_0024.InfoData.DcInputShift <-> InfoData/DcInputShift
//     PlcTask Inputs/GVL_iXlinker.EtherCAT_Master_ATxxxx.Beckhoff_ATH2xxx.Beckhoff_ATH2xxxEK1122.A_0009_ATH2050_0500_0024.InfoData.State <-> InfoData/State
//   PLC/PLC Instance <-> EtherCAT Master ATxxxx/Beckhoff ATH2xxx/Beckhoff ATH2xxxEK1122/A_0010(ATH2050-0501-0022)
//     PlcTask Inputs/GVL_iXlinker.EtherCAT_Master_ATxxxx.Beckhoff_ATH2xxx.Beckhoff_ATH2xxxEK1122.A_0010_ATH2050_0501_0022.CC_Inputs.Status <-> CC Inputs/Status
//     PlcTask Inputs/GVL_iXlinker.EtherCAT_Master_ATxxxx.Beckhoff_ATH2xxx.Beckhoff_ATH2xxxEK1122.A_0010_ATH2050_0501_0022.CC_Inputs.Current_actual_value_Ch[0] <-> CC Inputs/Current actual value Ch.1
//     PlcTask Inputs/GVL_iXlinker.EtherCAT_Master_ATxxxx.Beckhoff_ATH2xxx.Beckhoff_ATH2xxxEK1122.A_0010_ATH2050_0501_0022.CC_Inputs.Current_actual_value_Ch[1] <-> CC Inputs/Current actual value Ch.2
//     PlcTask Inputs/GVL_iXlinker.EtherCAT_Master_ATxxxx.Beckhoff_ATH2xxx.Beckhoff_ATH2xxxEK1122.A_0010_ATH2050_0501_0022.CC_Inputs.Current_actual_value_Ch[2] <-> CC Inputs/Current actual value Ch.3
//     PlcTask Inputs/GVL_iXlinker.EtherCAT_Master_ATxxxx.Beckhoff_ATH2xxx.Beckhoff_ATH2xxxEK1122.A_0010_ATH2050_0501_0022.CC_Inputs.Current_actual_value_Ch[3] <-> CC Inputs/Current actual value Ch.4
//     PlcTask Inputs/GVL_iXlinker.EtherCAT_Master_ATxxxx.Beckhoff_ATH2xxx.Beckhoff_ATH2xxxEK1122.A_0010_ATH2050_0501_0022.CC_Inputs.Current_actual_value_Ch[4] <-> CC Inputs/Current actual value Ch.5
//     PlcTask Inputs/GVL_iXlinker.EtherCAT_Master_ATxxxx.Beckhoff_ATH2xxx.Beckhoff_ATH2xxxEK1122.A_0010_ATH2050_0501_0022.CC_Inputs.Current_actual_value_Ch[5] <-> CC Inputs/Current actual value Ch.6
//     PlcTask Inputs/GVL_iXlinker.EtherCAT_Master_ATxxxx.Beckhoff_ATH2xxx.Beckhoff_ATH2xxxEK1122.A_0010_ATH2050_0501_0022.CC_Inputs.Current_actual_value_Ch[6] <-> CC Inputs/Current actual value Ch.7
//     PlcTask Inputs/GVL_iXlinker.EtherCAT_Master_ATxxxx.Beckhoff_ATH2xxx.Beckhoff_ATH2xxxEK1122.A_0010_ATH2050_0501_0022.CC_Inputs.Current_actual_value_Ch[7] <-> CC Inputs/Current actual value Ch.8
//     PlcTask Inputs/GVL_iXlinker.EtherCAT_Master_ATxxxx.Beckhoff_ATH2xxx.Beckhoff_ATH2xxxEK1122.A_0010_ATH2050_0501_0022.CC_Inputs.Current_actual_value_Ch[8] <-> CC Inputs/Current actual value Ch.9
//     PlcTask Inputs/GVL_iXlinker.EtherCAT_Master_ATxxxx.Beckhoff_ATH2xxx.Beckhoff_ATH2xxxEK1122.A_0010_ATH2050_0501_0022.CC_Inputs.Current_actual_value_Ch[9] <-> CC Inputs/Current actual value Ch.10
//     PlcTask Inputs/GVL_iXlinker.EtherCAT_Master_ATxxxx.Beckhoff_ATH2xxx.Beckhoff_ATH2xxxEK1122.A_0010_ATH2050_0501_0022.CC_Inputs.Current_actual_value_Ch[10] <-> CC Inputs/Current actual value Ch.11
//     PlcTask Inputs/GVL_iXlinker.EtherCAT_Master_ATxxxx.Beckhoff_ATH2xxx.Beckhoff_ATH2xxxEK1122.A_0010_ATH2050_0501_0022.CC_Inputs.Current_actual_value_Ch[11] <-> CC Inputs/Current actual value Ch.12
//     PlcTask Inputs/GVL_iXlinker.EtherCAT_Master_ATxxxx.Beckhoff_ATH2xxx.Beckhoff_ATH2xxxEK1122.A_0010_ATH2050_0501_0022.CC_Inputs.Current_actual_value_Ch[12] <-> CC Inputs/Current actual value Ch.13
//     PlcTask Inputs/GVL_iXlinker.EtherCAT_Master_ATxxxx.Beckhoff_ATH2xxx.Beckhoff_ATH2xxxEK1122.A_0010_ATH2050_0501_0022.CC_Inputs.Current_actual_value_Ch[13] <-> CC Inputs/Current actual value Ch.14
//     PlcTask Inputs/GVL_iXlinker.EtherCAT_Master_ATxxxx.Beckhoff_ATH2xxx.Beckhoff_ATH2xxxEK1122.A_0010_ATH2050_0501_0022.CC_Inputs.Current_actual_value_Ch[14] <-> CC Inputs/Current actual value Ch.15
//     PlcTask Outputs/GVL_iXlinker.EtherCAT_Master_ATxxxx.Beckhoff_ATH2xxx.Beckhoff_ATH2xxxEK1122.A_0010_ATH2050_0501_0022.CC_Outputs.Control <-> CC Outputs/Control
//     PlcTask Outputs/GVL_iXlinker.EtherCAT_Master_ATxxxx.Beckhoff_ATH2xxx.Beckhoff_ATH2xxxEK1122.A_0010_ATH2050_0501_0022.CC_Outputs.Current_setpoint_value_Ch[0] <-> CC Outputs/Current setpoint value Ch.1
//     PlcTask Outputs/GVL_iXlinker.EtherCAT_Master_ATxxxx.Beckhoff_ATH2xxx.Beckhoff_ATH2xxxEK1122.A_0010_ATH2050_0501_0022.CC_Outputs.Current_setpoint_value_Ch[1] <-> CC Outputs/Current setpoint value Ch.2
//     PlcTask Outputs/GVL_iXlinker.EtherCAT_Master_ATxxxx.Beckhoff_ATH2xxx.Beckhoff_ATH2xxxEK1122.A_0010_ATH2050_0501_0022.CC_Outputs.Current_setpoint_value_Ch[2] <-> CC Outputs/Current setpoint value Ch.3
//     PlcTask Outputs/GVL_iXlinker.EtherCAT_Master_ATxxxx.Beckhoff_ATH2xxx.Beckhoff_ATH2xxxEK1122.A_0010_ATH2050_0501_0022.CC_Outputs.Current_setpoint_value_Ch[3] <-> CC Outputs/Current setpoint value Ch.4
//     PlcTask Outputs/GVL_iXlinker.EtherCAT_Master_ATxxxx.Beckhoff_ATH2xxx.Beckhoff_ATH2xxxEK1122.A_0010_ATH2050_0501_0022.CC_Outputs.Current_setpoint_value_Ch[4] <-> CC Outputs/Current setpoint value Ch.5
//     PlcTask Outputs/GVL_iXlinker.EtherCAT_Master_ATxxxx.Beckhoff_ATH2xxx.Beckhoff_ATH2xxxEK1122.A_0010_ATH2050_0501_0022.CC_Outputs.Current_setpoint_value_Ch[5] <-> CC Outputs/Current setpoint value Ch.6
//     PlcTask Outputs/GVL_iXlinker.EtherCAT_Master_ATxxxx.Beckhoff_ATH2xxx.Beckhoff_ATH2xxxEK1122.A_0010_ATH2050_0501_0022.CC_Outputs.Current_setpoint_value_Ch[6] <-> CC Outputs/Current setpoint value Ch.7
//     PlcTask Outputs/GVL_iXlinker.EtherCAT_Master_ATxxxx.Beckhoff_ATH2xxx.Beckhoff_ATH2xxxEK1122.A_0010_ATH2050_0501_0022.CC_Outputs.Current_setpoint_value_Ch[7] <-> CC Outputs/Current setpoint value Ch.8
//     PlcTask Outputs/GVL_iXlinker.EtherCAT_Master_ATxxxx.Beckhoff_ATH2xxx.Beckhoff_ATH2xxxEK1122.A_0010_ATH2050_0501_0022.CC_Outputs.Current_setpoint_value_Ch[8] <-> CC Outputs/Current setpoint value Ch.9
//     PlcTask Outputs/GVL_iXlinker.EtherCAT_Master_ATxxxx.Beckhoff_ATH2xxx.Beckhoff_ATH2xxxEK1122.A_0010_ATH2050_0501_0022.CC_Outputs.Current_setpoint_value_Ch[9] <-> CC Outputs/Current setpoint value Ch.10
//     PlcTask Outputs/GVL_iXlinker.EtherCAT_Master_ATxxxx.Beckhoff_ATH2xxx.Beckhoff_ATH2xxxEK1122.A_0010_ATH2050_0501_0022.CC_Outputs.Current_setpoint_value_Ch[10] <-> CC Outputs/Current setpoint value Ch.11
//     PlcTask Outputs/GVL_iXlinker.EtherCAT_Master_ATxxxx.Beckhoff_ATH2xxx.Beckhoff_ATH2xxxEK1122.A_0010_ATH2050_0501_0022.CC_Outputs.Current_setpoint_value_Ch[11] <-> CC Outputs/Current setpoint value Ch.12
//     PlcTask Outputs/GVL_iXlinker.EtherCAT_Master_ATxxxx.Beckhoff_ATH2xxx.Beckhoff_ATH2xxxEK1122.A_0010_ATH2050_0501_0022.CC_Outputs.Current_setpoint_value_Ch[12] <-> CC Outputs/Current setpoint value Ch.13
//     PlcTask Outputs/GVL_iXlinker.EtherCAT_Master_ATxxxx.Beckhoff_ATH2xxx.Beckhoff_ATH2xxxEK1122.A_0010_ATH2050_0501_0022.CC_Outputs.Current_setpoint_value_Ch[13] <-> CC Outputs/Current setpoint value Ch.14
//     PlcTask Outputs/GVL_iXlinker.EtherCAT_Master_ATxxxx.Beckhoff_ATH2xxx.Beckhoff_ATH2xxxEK1122.A_0010_ATH2050_0501_0022.CC_Outputs.Current_setpoint_value_Ch[14] <-> CC Outputs/Current setpoint value Ch.15
//     PlcTask Inputs/GVL_iXlinker.EtherCAT_Master_ATxxxx.Beckhoff_ATH2xxx.Beckhoff_ATH2xxxEK1122.A_0010_ATH2050_0501_0022.WcState.WcState <-> WcState/WcState
//     PlcTask Inputs/GVL_iXlinker.EtherCAT_Master_ATxxxx.Beckhoff_ATH2xxx.Beckhoff_ATH2xxxEK1122.A_0010_ATH2050_0501_0022.WcState.InputToggle <-> WcState/InputToggle
//     PlcTask Inputs/GVL_iXlinker.EtherCAT_Master_ATxxxx.Beckhoff_ATH2xxx.Beckhoff_ATH2xxxEK1122.A_0010_ATH2050_0501_0022.InfoData.AdsAddr <-> InfoData/AdsAddr
//     PlcTask Inputs/GVL_iXlinker.EtherCAT_Master_ATxxxx.Beckhoff_ATH2xxx.Beckhoff_ATH2xxxEK1122.A_0010_ATH2050_0501_0022.InfoData.DcOutputShift <-> InfoData/DcOutputShift
//     PlcTask Inputs/GVL_iXlinker.EtherCAT_Master_ATxxxx.Beckhoff_ATH2xxx.Beckhoff_ATH2xxxEK1122.A_0010_ATH2050_0501_0022.InfoData.DcInputShift <-> InfoData/DcInputShift
//     PlcTask Inputs/GVL_iXlinker.EtherCAT_Master_ATxxxx.Beckhoff_ATH2xxx.Beckhoff_ATH2xxxEK1122.A_0010_ATH2050_0501_0022.InfoData.State <-> InfoData/State
//   PLC/PLC Instance <-> EtherCAT Master ATxxxx/Beckhoff ATH2xxx/Beckhoff ATH2xxxEK1122/A_0011(ATH2050-0501-0023)
//     PlcTask Inputs/GVL_iXlinker.EtherCAT_Master_ATxxxx.Beckhoff_ATH2xxx.Beckhoff_ATH2xxxEK1122.A_0011_ATH2050_0501_0023.CC_Inputs.Status <-> CC Inputs/Status
//     PlcTask Inputs/GVL_iXlinker.EtherCAT_Master_ATxxxx.Beckhoff_ATH2xxx.Beckhoff_ATH2xxxEK1122.A_0011_ATH2050_0501_0023.CC_Inputs.Current_actual_value_Ch[0] <-> CC Inputs/Current actual value Ch.1
//     PlcTask Inputs/GVL_iXlinker.EtherCAT_Master_ATxxxx.Beckhoff_ATH2xxx.Beckhoff_ATH2xxxEK1122.A_0011_ATH2050_0501_0023.CC_Inputs.Current_actual_value_Ch[1] <-> CC Inputs/Current actual value Ch.2
//     PlcTask Inputs/GVL_iXlinker.EtherCAT_Master_ATxxxx.Beckhoff_ATH2xxx.Beckhoff_ATH2xxxEK1122.A_0011_ATH2050_0501_0023.CC_Inputs.Current_actual_value_Ch[2] <-> CC Inputs/Current actual value Ch.3
//     PlcTask Inputs/GVL_iXlinker.EtherCAT_Master_ATxxxx.Beckhoff_ATH2xxx.Beckhoff_ATH2xxxEK1122.A_0011_ATH2050_0501_0023.CC_Inputs.Current_actual_value_Ch[3] <-> CC Inputs/Current actual value Ch.4
//     PlcTask Inputs/GVL_iXlinker.EtherCAT_Master_ATxxxx.Beckhoff_ATH2xxx.Beckhoff_ATH2xxxEK1122.A_0011_ATH2050_0501_0023.CC_Inputs.Current_actual_value_Ch[4] <-> CC Inputs/Current actual value Ch.5
//     PlcTask Inputs/GVL_iXlinker.EtherCAT_Master_ATxxxx.Beckhoff_ATH2xxx.Beckhoff_ATH2xxxEK1122.A_0011_ATH2050_0501_0023.CC_Inputs.Current_actual_value_Ch[5] <-> CC Inputs/Current actual value Ch.6
//     PlcTask Inputs/GVL_iXlinker.EtherCAT_Master_ATxxxx.Beckhoff_ATH2xxx.Beckhoff_ATH2xxxEK1122.A_0011_ATH2050_0501_0023.CC_Inputs.Current_actual_value_Ch[6] <-> CC Inputs/Current actual value Ch.7
//     PlcTask Inputs/GVL_iXlinker.EtherCAT_Master_ATxxxx.Beckhoff_ATH2xxx.Beckhoff_ATH2xxxEK1122.A_0011_ATH2050_0501_0023.CC_Inputs.Current_actual_value_Ch[7] <-> CC Inputs/Current actual value Ch.8
//     PlcTask Inputs/GVL_iXlinker.EtherCAT_Master_ATxxxx.Beckhoff_ATH2xxx.Beckhoff_ATH2xxxEK1122.A_0011_ATH2050_0501_0023.CC_Inputs.Current_actual_value_Ch[8] <-> CC Inputs/Current actual value Ch.9
//     PlcTask Inputs/GVL_iXlinker.EtherCAT_Master_ATxxxx.Beckhoff_ATH2xxx.Beckhoff_ATH2xxxEK1122.A_0011_ATH2050_0501_0023.CC_Inputs.Current_actual_value_Ch[9] <-> CC Inputs/Current actual value Ch.10
//     PlcTask Inputs/GVL_iXlinker.EtherCAT_Master_ATxxxx.Beckhoff_ATH2xxx.Beckhoff_ATH2xxxEK1122.A_0011_ATH2050_0501_0023.CC_Inputs.Current_actual_value_Ch[10] <-> CC Inputs/Current actual value Ch.11
//     PlcTask Inputs/GVL_iXlinker.EtherCAT_Master_ATxxxx.Beckhoff_ATH2xxx.Beckhoff_ATH2xxxEK1122.A_0011_ATH2050_0501_0023.CC_Inputs.Current_actual_value_Ch[11] <-> CC Inputs/Current actual value Ch.12
//     PlcTask Inputs/GVL_iXlinker.EtherCAT_Master_ATxxxx.Beckhoff_ATH2xxx.Beckhoff_ATH2xxxEK1122.A_0011_ATH2050_0501_0023.CC_Inputs.Current_actual_value_Ch[12] <-> CC Inputs/Current actual value Ch.13
//     PlcTask Inputs/GVL_iXlinker.EtherCAT_Master_ATxxxx.Beckhoff_ATH2xxx.Beckhoff_ATH2xxxEK1122.A_0011_ATH2050_0501_0023.CC_Inputs.Current_actual_value_Ch[13] <-> CC Inputs/Current actual value Ch.14
//     PlcTask Inputs/GVL_iXlinker.EtherCAT_Master_ATxxxx.Beckhoff_ATH2xxx.Beckhoff_ATH2xxxEK1122.A_0011_ATH2050_0501_0023.CC_Inputs.Current_actual_value_Ch[14] <-> CC Inputs/Current actual value Ch.15
//     PlcTask Outputs/GVL_iXlinker.EtherCAT_Master_ATxxxx.Beckhoff_ATH2xxx.Beckhoff_ATH2xxxEK1122.A_0011_ATH2050_0501_0023.CC_Outputs.Control <-> CC Outputs/Control
//     PlcTask Outputs/GVL_iXlinker.EtherCAT_Master_ATxxxx.Beckhoff_ATH2xxx.Beckhoff_ATH2xxxEK1122.A_0011_ATH2050_0501_0023.CC_Outputs.Current_setpoint_value_Ch[0] <-> CC Outputs/Current setpoint value Ch.1
//     PlcTask Outputs/GVL_iXlinker.EtherCAT_Master_ATxxxx.Beckhoff_ATH2xxx.Beckhoff_ATH2xxxEK1122.A_0011_ATH2050_0501_0023.CC_Outputs.Current_setpoint_value_Ch[1] <-> CC Outputs/Current setpoint value Ch.2
//     PlcTask Outputs/GVL_iXlinker.EtherCAT_Master_ATxxxx.Beckhoff_ATH2xxx.Beckhoff_ATH2xxxEK1122.A_0011_ATH2050_0501_0023.CC_Outputs.Current_setpoint_value_Ch[2] <-> CC Outputs/Current setpoint value Ch.3
//     PlcTask Outputs/GVL_iXlinker.EtherCAT_Master_ATxxxx.Beckhoff_ATH2xxx.Beckhoff_ATH2xxxEK1122.A_0011_ATH2050_0501_0023.CC_Outputs.Current_setpoint_value_Ch[3] <-> CC Outputs/Current setpoint value Ch.4
//     PlcTask Outputs/GVL_iXlinker.EtherCAT_Master_ATxxxx.Beckhoff_ATH2xxx.Beckhoff_ATH2xxxEK1122.A_0011_ATH2050_0501_0023.CC_Outputs.Current_setpoint_value_Ch[4] <-> CC Outputs/Current setpoint value Ch.5
//     PlcTask Outputs/GVL_iXlinker.EtherCAT_Master_ATxxxx.Beckhoff_ATH2xxx.Beckhoff_ATH2xxxEK1122.A_0011_ATH2050_0501_0023.CC_Outputs.Current_setpoint_value_Ch[5] <-> CC Outputs/Current setpoint value Ch.6
//     PlcTask Outputs/GVL_iXlinker.EtherCAT_Master_ATxxxx.Beckhoff_ATH2xxx.Beckhoff_ATH2xxxEK1122.A_0011_ATH2050_0501_0023.CC_Outputs.Current_setpoint_value_Ch[6] <-> CC Outputs/Current setpoint value Ch.7
//     PlcTask Outputs/GVL_iXlinker.EtherCAT_Master_ATxxxx.Beckhoff_ATH2xxx.Beckhoff_ATH2xxxEK1122.A_0011_ATH2050_0501_0023.CC_Outputs.Current_setpoint_value_Ch[7] <-> CC Outputs/Current setpoint value Ch.8
//     PlcTask Outputs/GVL_iXlinker.EtherCAT_Master_ATxxxx.Beckhoff_ATH2xxx.Beckhoff_ATH2xxxEK1122.A_0011_ATH2050_0501_0023.CC_Outputs.Current_setpoint_value_Ch[8] <-> CC Outputs/Current setpoint value Ch.9
//     PlcTask Outputs/GVL_iXlinker.EtherCAT_Master_ATxxxx.Beckhoff_ATH2xxx.Beckhoff_ATH2xxxEK1122.A_0011_ATH2050_0501_0023.CC_Outputs.Current_setpoint_value_Ch[9] <-> CC Outputs/Current setpoint value Ch.10
//     PlcTask Outputs/GVL_iXlinker.EtherCAT_Master_ATxxxx.Beckhoff_ATH2xxx.Beckhoff_ATH2xxxEK1122.A_0011_ATH2050_0501_0023.CC_Outputs.Current_setpoint_value_Ch[10] <-> CC Outputs/Current setpoint value Ch.11
//     PlcTask Outputs/GVL_iXlinker.EtherCAT_Master_ATxxxx.Beckhoff_ATH2xxx.Beckhoff_ATH2xxxEK1122.A_0011_ATH2050_0501_0023.CC_Outputs.Current_setpoint_value_Ch[11] <-> CC Outputs/Current setpoint value Ch.12
//     PlcTask Outputs/GVL_iXlinker.EtherCAT_Master_ATxxxx.Beckhoff_ATH2xxx.Beckhoff_ATH2xxxEK1122.A_0011_ATH2050_0501_0023.CC_Outputs.Current_setpoint_value_Ch[12] <-> CC Outputs/Current setpoint value Ch.13
//     PlcTask Outputs/GVL_iXlinker.EtherCAT_Master_ATxxxx.Beckhoff_ATH2xxx.Beckhoff_ATH2xxxEK1122.A_0011_ATH2050_0501_0023.CC_Outputs.Current_setpoint_value_Ch[13] <-> CC Outputs/Current setpoint value Ch.14
//     PlcTask Outputs/GVL_iXlinker.EtherCAT_Master_ATxxxx.Beckhoff_ATH2xxx.Beckhoff_ATH2xxxEK1122.A_0011_ATH2050_0501_0023.CC_Outputs.Current_setpoint_value_Ch[14] <-> CC Outputs/Current setpoint value Ch.15
//     PlcTask Inputs/GVL_iXlinker.EtherCAT_Master_ATxxxx.Beckhoff_ATH2xxx.Beckhoff_ATH2xxxEK1122.A_0011_ATH2050_0501_0023.WcState.WcState <-> WcState/WcState
//     PlcTask Inputs/GVL_iXlinker.EtherCAT_Master_ATxxxx.Beckhoff_ATH2xxx.Beckhoff_ATH2xxxEK1122.A_0011_ATH2050_0501_0023.WcState.InputToggle <-> WcState/InputToggle
//     PlcTask Inputs/GVL_iXlinker.EtherCAT_Master_ATxxxx.Beckhoff_ATH2xxx.Beckhoff_ATH2xxxEK1122.A_0011_ATH2050_0501_0023.InfoData.AdsAddr <-> InfoData/AdsAddr
//     PlcTask Inputs/GVL_iXlinker.EtherCAT_Master_ATxxxx.Beckhoff_ATH2xxx.Beckhoff_ATH2xxxEK1122.A_0011_ATH2050_0501_0023.InfoData.DcOutputShift <-> InfoData/DcOutputShift
//     PlcTask Inputs/GVL_iXlinker.EtherCAT_Master_ATxxxx.Beckhoff_ATH2xxx.Beckhoff_ATH2xxxEK1122.A_0011_ATH2050_0501_0023.InfoData.DcInputShift <-> InfoData/DcInputShift
//     PlcTask Inputs/GVL_iXlinker.EtherCAT_Master_ATxxxx.Beckhoff_ATH2xxx.Beckhoff_ATH2xxxEK1122.A_0011_ATH2050_0501_0023.InfoData.State <-> InfoData/State
//   PLC/PLC Instance <-> EtherCAT Master ATxxxx/Beckhoff ATH2xxx/Beckhoff ATH2xxxEK1122/A_0012(ATH2050-0501-0024)
//     PlcTask Inputs/GVL_iXlinker.EtherCAT_Master_ATxxxx.Beckhoff_ATH2xxx.Beckhoff_ATH2xxxEK1122.A_0012_ATH2050_0501_0024.CC_Inputs.Status <-> CC Inputs/Status
//     PlcTask Inputs/GVL_iXlinker.EtherCAT_Master_ATxxxx.Beckhoff_ATH2xxx.Beckhoff_ATH2xxxEK1122.A_0012_ATH2050_0501_0024.CC_Inputs.Current_actual_value_Ch[0] <-> CC Inputs/Current actual value Ch.1
//     PlcTask Inputs/GVL_iXlinker.EtherCAT_Master_ATxxxx.Beckhoff_ATH2xxx.Beckhoff_ATH2xxxEK1122.A_0012_ATH2050_0501_0024.CC_Inputs.Current_actual_value_Ch[1] <-> CC Inputs/Current actual value Ch.2
//     PlcTask Inputs/GVL_iXlinker.EtherCAT_Master_ATxxxx.Beckhoff_ATH2xxx.Beckhoff_ATH2xxxEK1122.A_0012_ATH2050_0501_0024.CC_Inputs.Current_actual_value_Ch[2] <-> CC Inputs/Current actual value Ch.3
//     PlcTask Inputs/GVL_iXlinker.EtherCAT_Master_ATxxxx.Beckhoff_ATH2xxx.Beckhoff_ATH2xxxEK1122.A_0012_ATH2050_0501_0024.CC_Inputs.Current_actual_value_Ch[3] <-> CC Inputs/Current actual value Ch.4
//     PlcTask Inputs/GVL_iXlinker.EtherCAT_Master_ATxxxx.Beckhoff_ATH2xxx.Beckhoff_ATH2xxxEK1122.A_0012_ATH2050_0501_0024.CC_Inputs.Current_actual_value_Ch[4] <-> CC Inputs/Current actual value Ch.5
//     PlcTask Inputs/GVL_iXlinker.EtherCAT_Master_ATxxxx.Beckhoff_ATH2xxx.Beckhoff_ATH2xxxEK1122.A_0012_ATH2050_0501_0024.CC_Inputs.Current_actual_value_Ch[5] <-> CC Inputs/Current actual value Ch.6
//     PlcTask Inputs/GVL_iXlinker.EtherCAT_Master_ATxxxx.Beckhoff_ATH2xxx.Beckhoff_ATH2xxxEK1122.A_0012_ATH2050_0501_0024.CC_Inputs.Current_actual_value_Ch[6] <-> CC Inputs/Current actual value Ch.7
//     PlcTask Inputs/GVL_iXlinker.EtherCAT_Master_ATxxxx.Beckhoff_ATH2xxx.Beckhoff_ATH2xxxEK1122.A_0012_ATH2050_0501_0024.CC_Inputs.Current_actual_value_Ch[7] <-> CC Inputs/Current actual value Ch.8
//     PlcTask Inputs/GVL_iXlinker.EtherCAT_Master_ATxxxx.Beckhoff_ATH2xxx.Beckhoff_ATH2xxxEK1122.A_0012_ATH2050_0501_0024.CC_Inputs.Current_actual_value_Ch[8] <-> CC Inputs/Current actual value Ch.9
//     PlcTask Inputs/GVL_iXlinker.EtherCAT_Master_ATxxxx.Beckhoff_ATH2xxx.Beckhoff_ATH2xxxEK1122.A_0012_ATH2050_0501_0024.CC_Inputs.Current_actual_value_Ch[9] <-> CC Inputs/Current actual value Ch.10
//     PlcTask Inputs/GVL_iXlinker.EtherCAT_Master_ATxxxx.Beckhoff_ATH2xxx.Beckhoff_ATH2xxxEK1122.A_0012_ATH2050_0501_0024.CC_Inputs.Current_actual_value_Ch[10] <-> CC Inputs/Current actual value Ch.11
//     PlcTask Inputs/GVL_iXlinker.EtherCAT_Master_ATxxxx.Beckhoff_ATH2xxx.Beckhoff_ATH2xxxEK1122.A_0012_ATH2050_0501_0024.CC_Inputs.Current_actual_value_Ch[11] <-> CC Inputs/Current actual value Ch.12
//     PlcTask Inputs/GVL_iXlinker.EtherCAT_Master_ATxxxx.Beckhoff_ATH2xxx.Beckhoff_ATH2xxxEK1122.A_0012_ATH2050_0501_0024.CC_Inputs.Current_actual_value_Ch[12] <-> CC Inputs/Current actual value Ch.13
//     PlcTask Inputs/GVL_iXlinker.EtherCAT_Master_ATxxxx.Beckhoff_ATH2xxx.Beckhoff_ATH2xxxEK1122.A_0012_ATH2050_0501_0024.CC_Inputs.Current_actual_value_Ch[13] <-> CC Inputs/Current actual value Ch.14
//     PlcTask Inputs/GVL_iXlinker.EtherCAT_Master_ATxxxx.Beckhoff_ATH2xxx.Beckhoff_ATH2xxxEK1122.A_0012_ATH2050_0501_0024.CC_Inputs.Current_actual_value_Ch[14] <-> CC Inputs/Current actual value Ch.15
//     PlcTask Outputs/GVL_iXlinker.EtherCAT_Master_ATxxxx.Beckhoff_ATH2xxx.Beckhoff_ATH2xxxEK1122.A_0012_ATH2050_0501_0024.CC_Outputs.Control <-> CC Outputs/Control
//     PlcTask Outputs/GVL_iXlinker.EtherCAT_Master_ATxxxx.Beckhoff_ATH2xxx.Beckhoff_ATH2xxxEK1122.A_0012_ATH2050_0501_0024.CC_Outputs.Current_setpoint_value_Ch[0] <-> CC Outputs/Current setpoint value Ch.1
//     PlcTask Outputs/GVL_iXlinker.EtherCAT_Master_ATxxxx.Beckhoff_ATH2xxx.Beckhoff_ATH2xxxEK1122.A_0012_ATH2050_0501_0024.CC_Outputs.Current_setpoint_value_Ch[1] <-> CC Outputs/Current setpoint value Ch.2
//     PlcTask Outputs/GVL_iXlinker.EtherCAT_Master_ATxxxx.Beckhoff_ATH2xxx.Beckhoff_ATH2xxxEK1122.A_0012_ATH2050_0501_0024.CC_Outputs.Current_setpoint_value_Ch[2] <-> CC Outputs/Current setpoint value Ch.3
//     PlcTask Outputs/GVL_iXlinker.EtherCAT_Master_ATxxxx.Beckhoff_ATH2xxx.Beckhoff_ATH2xxxEK1122.A_0012_ATH2050_0501_0024.CC_Outputs.Current_setpoint_value_Ch[3] <-> CC Outputs/Current setpoint value Ch.4
//     PlcTask Outputs/GVL_iXlinker.EtherCAT_Master_ATxxxx.Beckhoff_ATH2xxx.Beckhoff_ATH2xxxEK1122.A_0012_ATH2050_0501_0024.CC_Outputs.Current_setpoint_value_Ch[4] <-> CC Outputs/Current setpoint value Ch.5
//     PlcTask Outputs/GVL_iXlinker.EtherCAT_Master_ATxxxx.Beckhoff_ATH2xxx.Beckhoff_ATH2xxxEK1122.A_0012_ATH2050_0501_0024.CC_Outputs.Current_setpoint_value_Ch[5] <-> CC Outputs/Current setpoint value Ch.6
//     PlcTask Outputs/GVL_iXlinker.EtherCAT_Master_ATxxxx.Beckhoff_ATH2xxx.Beckhoff_ATH2xxxEK1122.A_0012_ATH2050_0501_0024.CC_Outputs.Current_setpoint_value_Ch[6] <-> CC Outputs/Current setpoint value Ch.7
//     PlcTask Outputs/GVL_iXlinker.EtherCAT_Master_ATxxxx.Beckhoff_ATH2xxx.Beckhoff_ATH2xxxEK1122.A_0012_ATH2050_0501_0024.CC_Outputs.Current_setpoint_value_Ch[7] <-> CC Outputs/Current setpoint value Ch.8
//     PlcTask Outputs/GVL_iXlinker.EtherCAT_Master_ATxxxx.Beckhoff_ATH2xxx.Beckhoff_ATH2xxxEK1122.A_0012_ATH2050_0501_0024.CC_Outputs.Current_setpoint_value_Ch[8] <-> CC Outputs/Current setpoint value Ch.9
//     PlcTask Outputs/GVL_iXlinker.EtherCAT_Master_ATxxxx.Beckhoff_ATH2xxx.Beckhoff_ATH2xxxEK1122.A_0012_ATH2050_0501_0024.CC_Outputs.Current_setpoint_value_Ch[9] <-> CC Outputs/Current setpoint value Ch.10
//     PlcTask Outputs/GVL_iXlinker.EtherCAT_Master_ATxxxx.Beckhoff_ATH2xxx.Beckhoff_ATH2xxxEK1122.A_0012_ATH2050_0501_0024.CC_Outputs.Current_setpoint_value_Ch[10] <-> CC Outputs/Current setpoint value Ch.11
//     PlcTask Outputs/GVL_iXlinker.EtherCAT_Master_ATxxxx.Beckhoff_ATH2xxx.Beckhoff_ATH2xxxEK1122.A_0012_ATH2050_0501_0024.CC_Outputs.Current_setpoint_value_Ch[11] <-> CC Outputs/Current setpoint value Ch.12
//     PlcTask Outputs/GVL_iXlinker.EtherCAT_Master_ATxxxx.Beckhoff_ATH2xxx.Beckhoff_ATH2xxxEK1122.A_0012_ATH2050_0501_0024.CC_Outputs.Current_setpoint_value_Ch[12] <-> CC Outputs/Current setpoint value Ch.13
//     PlcTask Outputs/GVL_iXlinker.EtherCAT_Master_ATxxxx.Beckhoff_ATH2xxx.Beckhoff_ATH2xxxEK1122.A_0012_ATH2050_0501_0024.CC_Outputs.Current_setpoint_value_Ch[13] <-> CC Outputs/Current setpoint value Ch.14
//     PlcTask Outputs/GVL_iXlinker.EtherCAT_Master_ATxxxx.Beckhoff_ATH2xxx.Beckhoff_ATH2xxxEK1122.A_0012_ATH2050_0501_0024.CC_Outputs.Current_setpoint_value_Ch[14] <-> CC Outputs/Current setpoint value Ch.15
//     PlcTask Inputs/GVL_iXlinker.EtherCAT_Master_ATxxxx.Beckhoff_ATH2xxx.Beckhoff_ATH2xxxEK1122.A_0012_ATH2050_0501_0024.WcState.WcState <-> WcState/WcState
//     PlcTask Inputs/GVL_iXlinker.EtherCAT_Master_ATxxxx.Beckhoff_ATH2xxx.Beckhoff_ATH2xxxEK1122.A_0012_ATH2050_0501_0024.WcState.InputToggle <-> WcState/InputToggle
//     PlcTask Inputs/GVL_iXlinker.EtherCAT_Master_ATxxxx.Beckhoff_ATH2xxx.Beckhoff_ATH2xxxEK1122.A_0012_ATH2050_0501_0024.InfoData.AdsAddr <-> InfoData/AdsAddr
//     PlcTask Inputs/GVL_iXlinker.EtherCAT_Master_ATxxxx.Beckhoff_ATH2xxx.Beckhoff_ATH2xxxEK1122.A_0012_ATH2050_0501_0024.InfoData.DcOutputShift <-> InfoData/DcOutputShift
//     PlcTask Inputs/GVL_iXlinker.EtherCAT_Master_ATxxxx.Beckhoff_ATH2xxx.Beckhoff_ATH2xxxEK1122.A_0012_ATH2050_0501_0024.InfoData.DcInputShift <-> InfoData/DcInputShift
//     PlcTask Inputs/GVL_iXlinker.EtherCAT_Master_ATxxxx.Beckhoff_ATH2xxx.Beckhoff_ATH2xxxEK1122.A_0012_ATH2050_0501_0024.InfoData.State <-> InfoData/State
//   PLC/PLC Instance <-> EtherCAT Master ATxxxx/Beckhoff ATH2xxx/A_0013(ATH2000-5250-0022)
//     PlcTask Inputs/GVL_iXlinker.EtherCAT_Master_ATxxxx.Beckhoff_ATH2xxx.A_0013_ATH2000_5250_0022.FB_Inputs.BinaryData <-> FB Inputs/BinaryData
//     PlcTask Outputs/GVL_iXlinker.EtherCAT_Master_ATxxxx.Beckhoff_ATH2xxx.A_0013_ATH2000_5250_0022.FB_Outputs.Control <-> FB Outputs/Control
//     PlcTask Inputs/GVL_iXlinker.EtherCAT_Master_ATxxxx.Beckhoff_ATH2xxx.A_0013_ATH2000_5250_0022.WcState.WcState <-> WcState/WcState
//     PlcTask Inputs/GVL_iXlinker.EtherCAT_Master_ATxxxx.Beckhoff_ATH2xxx.A_0013_ATH2000_5250_0022.WcState.InputToggle <-> WcState/InputToggle
//     PlcTask Inputs/GVL_iXlinker.EtherCAT_Master_ATxxxx.Beckhoff_ATH2xxx.A_0013_ATH2000_5250_0022.InfoData.DcOutputShift <-> InfoData/DcOutputShift
//     PlcTask Inputs/GVL_iXlinker.EtherCAT_Master_ATxxxx.Beckhoff_ATH2xxx.A_0013_ATH2000_5250_0022.InfoData.DcInputShift <-> InfoData/DcInputShift
//     PlcTask Inputs/GVL_iXlinker.EtherCAT_Master_ATxxxx.Beckhoff_ATH2xxx.A_0013_ATH2000_5250_0022.InfoData.State <-> InfoData/State
//   PLC/PLC Instance <-> EtherCAT_Master_ATxxxx
//     PlcTask Inputs/GVL_iXlinker.EtherCAT_Master_ATxxxx.SyncUnits._default._unreferenced.WcState.WcState <-> SyncUnits/<default>/<unreferenced>/WcState/WcState
//     PlcTask Inputs/GVL_iXlinker.EtherCAT_Master_ATxxxx.SyncUnits._default._unreferenced.InfoData.ObjectId <-> SyncUnits/<default>/<unreferenced>/InfoData/ObjectId
//     PlcTask Inputs/GVL_iXlinker.EtherCAT_Master_ATxxxx.SyncUnits._default._unreferenced.InfoData.State <-> SyncUnits/<default>/<unreferenced>/InfoData/State
//     PlcTask Inputs/GVL_iXlinker.EtherCAT_Master_ATxxxx.SyncUnits._default._unreferenced.InfoData.SlaveCount <-> SyncUnits/<default>/<unreferenced>/InfoData/SlaveCount
//     PlcTask Inputs/GVL_iXlinker.EtherCAT_Master_ATxxxx.SyncUnits._default.PlcTask.WcState.WcState <-> SyncUnits/<default>/PlcTask/WcState/WcState
//     PlcTask Inputs/GVL_iXlinker.EtherCAT_Master_ATxxxx.SyncUnits._default.PlcTask.InfoData.ObjectId <-> SyncUnits/<default>/PlcTask/InfoData/ObjectId
//     PlcTask Inputs/GVL_iXlinker.EtherCAT_Master_ATxxxx.SyncUnits._default.PlcTask.InfoData.State <-> SyncUnits/<default>/PlcTask/InfoData/State
//     PlcTask Inputs/GVL_iXlinker.EtherCAT_Master_ATxxxx.SyncUnits._default.PlcTask.InfoData.SlaveCount <-> SyncUnits/<default>/PlcTask/InfoData/SlaveCount
//     PlcTask Inputs/GVL_iXlinker.EtherCAT_Master_ATxxxx.Inputs.SlaveCount <-> Inputs/SlaveCount
//     PlcTask Inputs/GVL_iXlinker.EtherCAT_Master_ATxxxx.Inputs.DevState <-> Inputs/DevState
//     PlcTask Inputs/GVL_iXlinker.EtherCAT_Master_ATxxxx.Inputs.Frm{0..25}State <-> Inputs/Frm{0..25}State  (26 links)
//     PlcTask Inputs/GVL_iXlinker.EtherCAT_Master_ATxxxx.Inputs.Frm{0..25}WcState <-> Inputs/Frm{0..25}WcState  (26 links)
//     PlcTask Inputs/GVL_iXlinker.EtherCAT_Master_ATxxxx.Inputs.Frm{0..25}InputToggle <-> Inputs/Frm{0..25}InputToggle  (26 links)
//     PlcTask Outputs/GVL_iXlinker.EtherCAT_Master_ATxxxx.Outputs.DevCtrl <-> Outputs/DevCtrl
//     PlcTask Outputs/GVL_iXlinker.EtherCAT_Master_ATxxxx.Outputs.Frm{0..25}Ctrl <-> Outputs/Frm{0..25}Ctrl  (26 links)
//     PlcTask Outputs/GVL_iXlinker.EtherCAT_Master_ATxxxx.Outputs.Frm{0..25}WcCtrl <-> Outputs/Frm{0..25}WcCtrl  (26 links)
//     PlcTask Inputs/GVL_iXlinker.EtherCAT_Master_ATxxxx.InfoData.ChangeCount <-> InfoData/ChangeCount
//     PlcTask Inputs/GVL_iXlinker.EtherCAT_Master_ATxxxx.InfoData.DevId <-> InfoData/DevId
//     PlcTask Inputs/GVL_iXlinker.EtherCAT_Master_ATxxxx.InfoData.AmsNetId <-> InfoData/AmsNetId
//     PlcTask Inputs/GVL_iXlinker.EtherCAT_Master_ATxxxx.InfoData.CfgSlaveCount <-> InfoData/CfgSlaveCount
//     PlcTask Inputs/GVL_iXlinker.EtherCAT_Master_ATxxxx.InfoData.DcToTcTimeOffset <-> InfoData/DcToTcTimeOffset
//     PlcTask Inputs/GVL_iXlinker.EtherCAT_Master_ATxxxx.InfoData.DcToExtTimeOffset <-> InfoData/DcToExtTimeOffset

CONFIGURATION PLC
    RESOURCE PLC ON TwinCAT3
        TASK PlcTask(INTERVAL := T#10ms, PRIORITY := 20);
        PROGRAM MAIN WITH PlcTask : MAIN;
    END_RESOURCE
END_CONFIGURATION

// ---- DUTs/IO/PDOs/InfoData_6F19DB2B.TcDUT
{attribute 'GeneratedUsingTerminal: EK1100-0000-0018'}
{attribute addProperty BoxType "EK1100-0000-0018"}
{attribute addProperty Id "StateAT %I*UINT2"}
{attribute addProperty CRC "1863965483"}
{attribute addProperty Size "2"}
TYPE InfoData_6F19DB2B :
STRUCT
	{attribute addProperty Name "State"}
	State AT %I* : UINT;
END_STRUCT
END_TYPE

// ---- DUTs/IO/PDOs/CC_Inputs_2C1C9EE0.TcDUT
{attribute 'GeneratedUsingTerminal: AT2020-0250-0019'}
{attribute addProperty BoxType "AT2020-0250-0019"}
{attribute addProperty Id "StatusAT %I*UINT2Current_actual_value_ChAT %I*ARRAY[0..14] OF INT30"}
{attribute addProperty CRC "4120755276"}
{attribute addProperty Size "32"}
TYPE CC_Inputs_2C1C9EE0 EXTENDS InputBase_8311D824 :
STRUCT
	{attribute addProperty Name "Status"}
	Status AT %I* : UINT;
	{attribute addProperty Name "Current_actual_value_Ch"}
	Current_actual_value_Ch AT %I* : ARRAY[0..14] OF INT;
END_STRUCT
END_TYPE

// ---- DUTs/IO/PDOs/CC_Outputs_69F9BE14.TcDUT
{attribute 'GeneratedUsingTerminal: AT2020-0250-0019'}
{attribute addProperty BoxType "AT2020-0250-0019"}
{attribute addProperty Id "ControlAT %Q*UINT2Current_setpoint_value_ChAT %Q*ARRAY[0..14] OF INT30"}
{attribute addProperty CRC "3100183749"}
{attribute addProperty Size "32"}
TYPE CC_Outputs_69F9BE14 EXTENDS OutputBase_10CEE7DE :
STRUCT
	{attribute addProperty Name "Control"}
	Control AT %Q* : UINT;
	{attribute addProperty Name "Current_setpoint_value_Ch"}
	Current_setpoint_value_Ch AT %Q* : ARRAY[0..14] OF INT;
END_STRUCT
END_TYPE

// ---- DUTs/IO/PDOs/WcState_9091E0EB.TcDUT
{attribute 'GeneratedUsingTerminal: AT2020-0250-0019'}
{attribute addProperty BoxType "AT2020-0250-0019"}
{attribute addProperty Id "WcStateAT %I*BOOL1InputToggleAT %I*BOOL1"}
{attribute addProperty CRC "2425479403"}
{attribute addProperty Size "2"}
TYPE WcState_9091E0EB :
STRUCT
	{attribute addProperty Name "WcState"}
	WcState AT %I* : BOOL;
	{attribute addProperty Name "InputToggle"}
	InputToggle AT %I* : BOOL;
END_STRUCT
END_TYPE

// ---- DUTs/IO/PDOs/InfoData_BEF6B88E.TcDUT
{attribute 'GeneratedUsingTerminal: AT2020-0250-0019'}
{attribute addProperty BoxType "AT2020-0250-0019"}
{attribute addProperty Id "AdsAddrAT %I*AMSADDR8DcOutputShiftAT %I*DINT4DcInputShiftAT %I*DINT4StateAT %I*UINT2"}
{attribute addProperty CRC "3203840142"}
{attribute addProperty Size "18"}
TYPE InfoData_BEF6B88E EXTENDS InputBase_8311D824 :
STRUCT
	{attribute addProperty Name "AdsAddr"}
	AdsAddr AT %I* : AMSADDR;
	{attribute addProperty Name "DcOutputShift"}
	DcOutputShift AT %I* : DINT;
	{attribute addProperty Name "DcInputShift"}
	DcInputShift AT %I* : DINT;
	{attribute addProperty Name "State"}
	State AT %I* : UINT;
END_STRUCT
END_TYPE

// ---- DUTs/IO/PDOs/FB_Inputs_4BC4AA01.TcDUT
{attribute 'GeneratedUsingTerminal: AT2050-5500-0018'}
{attribute addProperty BoxType "AT2050-5500-0018"}
{attribute addProperty Id "StatusAT %I*UINT2Value_ChannelAT %I*ARRAY[0..31] OF INT64"}
{attribute addProperty CRC "3217050683"}
{attribute addProperty Size "66"}
TYPE FB_Inputs_4BC4AA01 EXTENDS InputBase_8311D824 :
STRUCT
	{attribute addProperty Name "Status"}
	Status AT %I* : UINT;
	{attribute addProperty Name "Value_Channel"}
	Value_Channel AT %I* : ARRAY[0..31] OF INT;
END_STRUCT
END_TYPE

// ---- DUTs/IO/PDOs/FB_Outputs_DAFD38E0.TcDUT
{attribute 'GeneratedUsingTerminal: AT2050-5500-0018'}
{attribute addProperty BoxType "AT2050-5500-0018"}
{attribute addProperty Id "ControlAT %Q*UINT2"}
{attribute addProperty CRC "3674028256"}
{attribute addProperty Size "2"}
TYPE FB_Outputs_DAFD38E0 EXTENDS OutputBase_10CEE7DE :
STRUCT
	{attribute addProperty Name "Control"}
	Control AT %Q* : UINT;
END_STRUCT
END_TYPE

// ---- DUTs/IO/PDOs/InfoData_A7436BC6.TcDUT
{attribute 'GeneratedUsingTerminal: AT2050-5500-0018'}
{attribute addProperty BoxType "AT2050-5500-0018"}
{attribute addProperty Id "DcOutputShiftAT %I*DINT4DcInputShiftAT %I*DINT4StateAT %I*UINT2"}
{attribute addProperty CRC "2806213574"}
{attribute addProperty Size "10"}
TYPE InfoData_A7436BC6 EXTENDS InputBase_8311D824 :
STRUCT
	{attribute addProperty Name "DcOutputShift"}
	DcOutputShift AT %I* : DINT;
	{attribute addProperty Name "DcInputShift"}
	DcInputShift AT %I* : DINT;
	{attribute addProperty Name "State"}
	State AT %I* : UINT;
END_STRUCT
END_TYPE

// ---- DUTs/IO/PDOs/CC_Inputs_14_Ch_F1B79554.TcDUT
{attribute 'GeneratedUsingTerminal: AT2000-0233-0022'}
{attribute addProperty BoxType "AT2000-0233-0022"}
{attribute addProperty Id "StatusAT %I*UINT2Current_actual_value_ChAT %I*ARRAY[0..13] OF INT28"}
{attribute addProperty CRC "3830004940"}
{attribute addProperty Size "30"}
TYPE CC_Inputs_14_Ch_F1B79554 EXTENDS InputBase_8311D824 :
STRUCT
	{attribute addProperty Name "Status"}
	Status AT %I* : UINT;
	{attribute addProperty Name "Current_actual_value_Ch"}
	Current_actual_value_Ch AT %I* : ARRAY[0..13] OF INT;
END_STRUCT
END_TYPE

// ---- DUTs/IO/PDOs/CC_Outputs_14_Ch_45965511.TcDUT
{attribute 'GeneratedUsingTerminal: AT2000-0233-0022'}
{attribute addProperty BoxType "AT2000-0233-0022"}
{attribute addProperty Id "ControlAT %Q*UINT2Current_setpoint_value_ChAT %Q*ARRAY[0..13] OF INT28"}
{attribute addProperty CRC "2837285957"}
{attribute addProperty Size "30"}
TYPE CC_Outputs_14_Ch_45965511 EXTENDS OutputBase_10CEE7DE :
STRUCT
	{attribute addProperty Name "Control"}
	Control AT %Q* : UINT;
	{attribute addProperty Name "Current_setpoint_value_Ch"}
	Current_setpoint_value_Ch AT %Q* : ARRAY[0..13] OF INT;
END_STRUCT
END_TYPE

// ---- DUTs/IO/PDOs/FB_Inputs_39145651.TcDUT
{attribute 'GeneratedUsingTerminal: ATH2050-5501-0022'}
{attribute addProperty BoxType "ATH2050-5501-0022"}
{attribute addProperty Id "BinaryDataAT %I*ARRAY [0..55] OF BYTE0"}
{attribute addProperty CRC "957634129"}
{attribute addProperty Size "0"}
TYPE FB_Inputs_39145651 EXTENDS InputBase_8311D824 :
STRUCT
	{attribute addProperty Name "BinaryData"}
	BinaryData AT %I* : ARRAY [0..55] OF BYTE;
END_STRUCT
END_TYPE

// ---- DUTs/IO/PDOs/FB_Inputs_01C60045.TcDUT
{attribute 'GeneratedUsingTerminal: ATH2040-5250-0022'}
{attribute addProperty BoxType "ATH2040-5250-0022"}
{attribute addProperty Id "BinaryDataAT %I*ARRAY [0..59] OF BYTE0"}
{attribute addProperty CRC "29753413"}
{attribute addProperty Size "0"}
TYPE FB_Inputs_01C60045 EXTENDS InputBase_8311D824 :
STRUCT
	{attribute addProperty Name "BinaryData"}
	BinaryData AT %I* : ARRAY [0..59] OF BYTE;
END_STRUCT
END_TYPE

// ---- DUTs/IO/PDOs/FB_Inputs_2D665851.TcDUT
{attribute 'GeneratedUsingTerminal: ATH2000-5250-0022'}
{attribute addProperty BoxType "ATH2000-5250-0022"}
{attribute addProperty Id "BinaryDataAT %I*ARRAY [0..63] OF BYTE0"}
{attribute addProperty CRC "761682001"}
{attribute addProperty Size "0"}
TYPE FB_Inputs_2D665851 EXTENDS InputBase_8311D824 :
STRUCT
	{attribute addProperty Name "BinaryData"}
	BinaryData AT %I* : ARRAY [0..63] OF BYTE;
END_STRUCT
END_TYPE

// ---- DUTs/IO/PDOs/InfoData_E68C61CD.TcDUT
{attribute 'GeneratedUsingTerminal: IODEVICETYPE_ETHERCATPROT'}
{attribute addProperty BoxType "IODEVICETYPE_ETHERCATPROT"}
{attribute addProperty Id "ChangeCountAT %I*UINT2DevIdAT %I*UINT2AmsNetIdAT %I*AMSNETID6CfgSlaveCountAT %I*UINT2DcToTcTimeOffsetAT %I*LINT8DcToExtTimeOffsetAT %I*LINT8"}
{attribute addProperty CRC "3867959757"}
{attribute addProperty Size "28"}
TYPE InfoData_E68C61CD EXTENDS InputBase_8311D824 :
STRUCT
	{attribute addProperty Name "ChangeCount"}
	ChangeCount AT %I* : UINT;
	{attribute addProperty Name "DevId"}
	DevId AT %I* : UINT;
	{attribute addProperty Name "AmsNetId"}
	AmsNetId AT %I* : AMSNETID;
	{attribute addProperty Name "CfgSlaveCount"}
	CfgSlaveCount AT %I* : UINT;
	{attribute addProperty Name "DcToTcTimeOffset"}
	DcToTcTimeOffset AT %I* : LINT;
	{attribute addProperty Name "DcToExtTimeOffset"}
	DcToExtTimeOffset AT %I* : LINT;
END_STRUCT
END_TYPE

// ---- DUTs/IO/PDOs/WcState_0B2B16F9.TcDUT
{attribute 'GeneratedUsingTerminal: IODEVICETYPE_ETHERCATPROT'}
{attribute addProperty BoxType "IODEVICETYPE_ETHERCATPROT"}
{attribute addProperty Id "WcStateAT %I*BOOL1"}
{attribute addProperty CRC "187373305"}
{attribute addProperty Size "1"}
TYPE WcState_0B2B16F9 :
STRUCT
	{attribute addProperty Name "WcState"}
	WcState AT %I* : BOOL;
END_STRUCT
END_TYPE

// ---- DUTs/IO/PDOs/InfoData_2A97D6CF.TcDUT
{attribute 'GeneratedUsingTerminal: IODEVICETYPE_ETHERCATPROT'}
{attribute addProperty BoxType "IODEVICETYPE_ETHERCATPROT"}
{attribute addProperty Id "ObjectIdAT %I*OTCID4StateAT %I*UINT2SlaveCountAT %I*UINT2"}
{attribute addProperty CRC "714593999"}
{attribute addProperty Size "8"}
TYPE InfoData_2A97D6CF EXTENDS InputBase_8311D824 :
STRUCT
	{attribute addProperty Name "ObjectId"}
	ObjectId AT %I* : OTCID;
	{attribute addProperty Name "State"}
	State AT %I* : UINT;
	{attribute addProperty Name "SlaveCount"}
	SlaveCount AT %I* : UINT;
END_STRUCT
END_TYPE

// ---- DUTs/IO/PDOs/Inputs_25A0042B.TcDUT
{attribute 'GeneratedUsingTerminal: IODEVICETYPE_ETHERCATPROT'}
{attribute addProperty BoxType "IODEVICETYPE_ETHERCATPROT"}
{attribute addProperty Id "SlaveCountAT %I*UINT2DevStateAT %I*UINT2Frm0StateAT %I*UINT2Frm0WcStateAT %I*UINT2Frm0InputToggleAT %I*UINT2Frm1StateAT %I*UINT2Frm1WcStateAT %I*UINT2Frm1InputToggleAT %I*UINT2Frm2StateAT %I*UINT2Frm2WcStateAT %I*UINT2Frm2InputToggleAT %I*UINT2Frm3StateAT %I*UINT2Frm3WcStateAT %I*UINT2Frm3InputToggleAT %I*UINT2Frm4StateAT %I*UINT2Frm4WcStateAT %I*UINT2Frm4InputToggleAT %I*UINT2Frm5StateAT %I*UINT2Frm5WcStateAT %I*UINT2Frm5InputToggleAT %I*UINT2Frm6StateAT %I*UINT2Frm6WcStateAT %I*UINT2Frm6InputToggleAT %I*UINT2Frm7StateAT %I*UINT2Frm7WcStateAT %I*UINT2Frm7InputToggleAT %I*UINT2Frm8StateAT %I*UINT2Frm8WcStateAT %I*UINT2Frm8InputToggleAT %I*UINT2Frm9StateAT %I*UINT2Frm9WcStateAT %I*UINT2Frm9InputToggleAT %I*UINT2Frm10StateAT %I*UINT2Frm10WcStateAT %I*UINT2Frm10InputToggleAT %I*UINT2Frm11StateAT %I*UINT2Frm11WcStateAT %I*UINT2Frm11InputToggleAT %I*UINT2Frm12StateAT %I*UINT2Frm12WcStateAT %I*UINT2Frm12InputToggleAT %I*UINT2Frm13StateAT %I*UINT2Frm13WcStateAT %I*UINT2Frm13InputToggleAT %I*UINT2Frm14StateAT %I*UINT2Frm14WcStateAT %I*UINT2Frm14InputToggleAT %I*UINT2Frm15StateAT %I*UINT2Frm15WcStateAT %I*UINT2Frm15InputToggleAT %I*UINT2Frm16StateAT %I*UINT2Frm16WcStateAT %I*UINT2Frm16InputToggleAT %I*UINT2Frm17StateAT %I*UINT2Frm17WcStateAT %I*UINT2Frm17InputToggleAT %I*UINT2Frm18StateAT %I*UINT2Frm18WcStateAT %I*UINT2Frm18InputToggleAT %I*UINT2Frm19StateAT %I*UINT2Frm19WcStateAT %I*UINT2Frm19InputToggleAT %I*UINT2Frm20StateAT %I*UINT2Frm20WcStateAT %I*UINT2Frm20InputToggleAT %I*UINT2Frm21StateAT %I*UINT2Frm21WcStateAT %I*UINT2Frm21InputToggleAT %I*UINT2Frm22StateAT %I*UINT2Frm22WcStateAT %I*UINT2Frm22InputToggleAT %I*UINT2Frm23StateAT %I*UINT2Frm23WcStateAT %I*UINT2Frm23InputToggleAT %I*UINT2Frm24StateAT %I*UINT2Frm24WcStateAT %I*UINT2Frm24InputToggleAT %I*UINT2Frm25StateAT %I*UINT2Frm25WcStateAT %I*UINT2Frm25InputToggleAT %I*UINT2"}
{attribute addProperty CRC "631243819"}
{attribute addProperty Size "160"}
TYPE Inputs_25A0042B EXTENDS InputBase_8311D824 :
STRUCT
	{attribute addProperty Name "SlaveCount"}
	SlaveCount AT %I* : UINT;
	{attribute addProperty Name "DevState"}
	DevState AT %I* : UINT;
	{attribute addProperty Name "Frm0State"}
	Frm0State AT %I* : UINT;
	{attribute addProperty Name "Frm0WcState"}
	Frm0WcState AT %I* : UINT;
	{attribute addProperty Name "Frm0InputToggle"}
	Frm0InputToggle AT %I* : UINT;
	{attribute addProperty Name "Frm1State"}
	Frm1State AT %I* : UINT;
	{attribute addProperty Name "Frm1WcState"}
	Frm1WcState AT %I* : UINT;
	{attribute addProperty Name "Frm1InputToggle"}
	Frm1InputToggle AT %I* : UINT;
	{attribute addProperty Name "Frm2State"}
	Frm2State AT %I* : UINT;
	{attribute addProperty Name "Frm2WcState"}
	Frm2WcState AT %I* : UINT;
	{attribute addProperty Name "Frm2InputToggle"}
	Frm2InputToggle AT %I* : UINT;
	{attribute addProperty Name "Frm3State"}
	Frm3State AT %I* : UINT;
	{attribute addProperty Name "Frm3WcState"}
	Frm3WcState AT %I* : UINT;
	{attribute addProperty Name "Frm3InputToggle"}
	Frm3InputToggle AT %I* : UINT;
	{attribute addProperty Name "Frm4State"}
	Frm4State AT %I* : UINT;
	{attribute addProperty Name "Frm4WcState"}
	Frm4WcState AT %I* : UINT;
	{attribute addProperty Name "Frm4InputToggle"}
	Frm4InputToggle AT %I* : UINT;
	{attribute addProperty Name "Frm5State"}
	Frm5State AT %I* : UINT;
	{attribute addProperty Name "Frm5WcState"}
	Frm5WcState AT %I* : UINT;
	{attribute addProperty Name "Frm5InputToggle"}
	Frm5InputToggle AT %I* : UINT;
	{attribute addProperty Name "Frm6State"}
	Frm6State AT %I* : UINT;
	{attribute addProperty Name "Frm6WcState"}
	Frm6WcState AT %I* : UINT;
	{attribute addProperty Name "Frm6InputToggle"}
	Frm6InputToggle AT %I* : UINT;
	{attribute addProperty Name "Frm7State"}
	Frm7State AT %I* : UINT;
	{attribute addProperty Name "Frm7WcState"}
	Frm7WcState AT %I* : UINT;
	{attribute addProperty Name "Frm7InputToggle"}
	Frm7InputToggle AT %I* : UINT;
	{attribute addProperty Name "Frm8State"}
	Frm8State AT %I* : UINT;
	{attribute addProperty Name "Frm8WcState"}
	Frm8WcState AT %I* : UINT;
	{attribute addProperty Name "Frm8InputToggle"}
	Frm8InputToggle AT %I* : UINT;
	{attribute addProperty Name "Frm9State"}
	Frm9State AT %I* : UINT;
	{attribute addProperty Name "Frm9WcState"}
	Frm9WcState AT %I* : UINT;
	{attribute addProperty Name "Frm9InputToggle"}
	Frm9InputToggle AT %I* : UINT;
	{attribute addProperty Name "Frm10State"}
	Frm10State AT %I* : UINT;
	{attribute addProperty Name "Frm10WcState"}
	Frm10WcState AT %I* : UINT;
	{attribute addProperty Name "Frm10InputToggle"}
	Frm10InputToggle AT %I* : UINT;
	{attribute addProperty Name "Frm11State"}
	Frm11State AT %I* : UINT;
	{attribute addProperty Name "Frm11WcState"}
	Frm11WcState AT %I* : UINT;
	{attribute addProperty Name "Frm11InputToggle"}
	Frm11InputToggle AT %I* : UINT;
	{attribute addProperty Name "Frm12State"}
	Frm12State AT %I* : UINT;
	{attribute addProperty Name "Frm12WcState"}
	Frm12WcState AT %I* : UINT;
	{attribute addProperty Name "Frm12InputToggle"}
	Frm12InputToggle AT %I* : UINT;
	{attribute addProperty Name "Frm13State"}
	Frm13State AT %I* : UINT;
	{attribute addProperty Name "Frm13WcState"}
	Frm13WcState AT %I* : UINT;
	{attribute addProperty Name "Frm13InputToggle"}
	Frm13InputToggle AT %I* : UINT;
	{attribute addProperty Name "Frm14State"}
	Frm14State AT %I* : UINT;
	{attribute addProperty Name "Frm14WcState"}
	Frm14WcState AT %I* : UINT;
	{attribute addProperty Name "Frm14InputToggle"}
	Frm14InputToggle AT %I* : UINT;
	{attribute addProperty Name "Frm15State"}
	Frm15State AT %I* : UINT;
	{attribute addProperty Name "Frm15WcState"}
	Frm15WcState AT %I* : UINT;
	{attribute addProperty Name "Frm15InputToggle"}
	Frm15InputToggle AT %I* : UINT;
	{attribute addProperty Name "Frm16State"}
	Frm16State AT %I* : UINT;
	{attribute addProperty Name "Frm16WcState"}
	Frm16WcState AT %I* : UINT;
	{attribute addProperty Name "Frm16InputToggle"}
	Frm16InputToggle AT %I* : UINT;
	{attribute addProperty Name "Frm17State"}
	Frm17State AT %I* : UINT;
	{attribute addProperty Name "Frm17WcState"}
	Frm17WcState AT %I* : UINT;
	{attribute addProperty Name "Frm17InputToggle"}
	Frm17InputToggle AT %I* : UINT;
	{attribute addProperty Name "Frm18State"}
	Frm18State AT %I* : UINT;
	{attribute addProperty Name "Frm18WcState"}
	Frm18WcState AT %I* : UINT;
	{attribute addProperty Name "Frm18InputToggle"}
	Frm18InputToggle AT %I* : UINT;
	{attribute addProperty Name "Frm19State"}
	Frm19State AT %I* : UINT;
	{attribute addProperty Name "Frm19WcState"}
	Frm19WcState AT %I* : UINT;
	{attribute addProperty Name "Frm19InputToggle"}
	Frm19InputToggle AT %I* : UINT;
	{attribute addProperty Name "Frm20State"}
	Frm20State AT %I* : UINT;
	{attribute addProperty Name "Frm20WcState"}
	Frm20WcState AT %I* : UINT;
	{attribute addProperty Name "Frm20InputToggle"}
	Frm20InputToggle AT %I* : UINT;
	{attribute addProperty Name "Frm21State"}
	Frm21State AT %I* : UINT;
	{attribute addProperty Name "Frm21WcState"}
	Frm21WcState AT %I* : UINT;
	{attribute addProperty Name "Frm21InputToggle"}
	Frm21InputToggle AT %I* : UINT;
	{attribute addProperty Name "Frm22State"}
	Frm22State AT %I* : UINT;
	{attribute addProperty Name "Frm22WcState"}
	Frm22WcState AT %I* : UINT;
	{attribute addProperty Name "Frm22InputToggle"}
	Frm22InputToggle AT %I* : UINT;
	{attribute addProperty Name "Frm23State"}
	Frm23State AT %I* : UINT;
	{attribute addProperty Name "Frm23WcState"}
	Frm23WcState AT %I* : UINT;
	{attribute addProperty Name "Frm23InputToggle"}
	Frm23InputToggle AT %I* : UINT;
	{attribute addProperty Name "Frm24State"}
	Frm24State AT %I* : UINT;
	{attribute addProperty Name "Frm24WcState"}
	Frm24WcState AT %I* : UINT;
	{attribute addProperty Name "Frm24InputToggle"}
	Frm24InputToggle AT %I* : UINT;
	{attribute addProperty Name "Frm25State"}
	Frm25State AT %I* : UINT;
	{attribute addProperty Name "Frm25WcState"}
	Frm25WcState AT %I* : UINT;
	{attribute addProperty Name "Frm25InputToggle"}
	Frm25InputToggle AT %I* : UINT;
END_STRUCT
END_TYPE

// ---- DUTs/IO/PDOs/Outputs_2397A10E.TcDUT
{attribute 'GeneratedUsingTerminal: IODEVICETYPE_ETHERCATPROT'}
{attribute addProperty BoxType "IODEVICETYPE_ETHERCATPROT"}
{attribute addProperty Id "DevCtrlAT %Q*UINT2Frm0CtrlAT %Q*UINT2Frm0WcCtrlAT %Q*UINT2Frm1CtrlAT %Q*UINT2Frm1WcCtrlAT %Q*UINT2Frm2CtrlAT %Q*UINT2Frm2WcCtrlAT %Q*UINT2Frm3CtrlAT %Q*UINT2Frm3WcCtrlAT %Q*UINT2Frm4CtrlAT %Q*UINT2Frm4WcCtrlAT %Q*UINT2Frm5CtrlAT %Q*UINT2Frm5WcCtrlAT %Q*UINT2Frm6CtrlAT %Q*UINT2Frm6WcCtrlAT %Q*UINT2Frm7CtrlAT %Q*UINT2Frm7WcCtrlAT %Q*UINT2Frm8CtrlAT %Q*UINT2Frm8WcCtrlAT %Q*UINT2Frm9CtrlAT %Q*UINT2Frm9WcCtrlAT %Q*UINT2Frm10CtrlAT %Q*UINT2Frm10WcCtrlAT %Q*UINT2Frm11CtrlAT %Q*UINT2Frm11WcCtrlAT %Q*UINT2Frm12CtrlAT %Q*UINT2Frm12WcCtrlAT %Q*UINT2Frm13CtrlAT %Q*UINT2Frm13WcCtrlAT %Q*UINT2Frm14CtrlAT %Q*UINT2Frm14WcCtrlAT %Q*UINT2Frm15CtrlAT %Q*UINT2Frm15WcCtrlAT %Q*UINT2Frm16CtrlAT %Q*UINT2Frm16WcCtrlAT %Q*UINT2Frm17CtrlAT %Q*UINT2Frm17WcCtrlAT %Q*UINT2Frm18CtrlAT %Q*UINT2Frm18WcCtrlAT %Q*UINT2Frm19CtrlAT %Q*UINT2Frm19WcCtrlAT %Q*UINT2Frm20CtrlAT %Q*UINT2Frm20WcCtrlAT %Q*UINT2Frm21CtrlAT %Q*UINT2Frm21WcCtrlAT %Q*UINT2Frm22CtrlAT %Q*UINT2Frm22WcCtrlAT %Q*UINT2Frm23CtrlAT %Q*UINT2Frm23WcCtrlAT %Q*UINT2Frm24CtrlAT %Q*UINT2Frm24WcCtrlAT %Q*UINT2Frm25CtrlAT %Q*UINT2Frm25WcCtrlAT %Q*UINT2"}
{attribute addProperty CRC "597139726"}
{attribute addProperty Size "106"}
TYPE Outputs_2397A10E EXTENDS OutputBase_10CEE7DE :
STRUCT
	{attribute addProperty Name "DevCtrl"}
	DevCtrl AT %Q* : UINT;
	{attribute addProperty Name "Frm0Ctrl"}
	Frm0Ctrl AT %Q* : UINT;
	{attribute addProperty Name "Frm0WcCtrl"}
	Frm0WcCtrl AT %Q* : UINT;
	{attribute addProperty Name "Frm1Ctrl"}
	Frm1Ctrl AT %Q* : UINT;
	{attribute addProperty Name "Frm1WcCtrl"}
	Frm1WcCtrl AT %Q* : UINT;
	{attribute addProperty Name "Frm2Ctrl"}
	Frm2Ctrl AT %Q* : UINT;
	{attribute addProperty Name "Frm2WcCtrl"}
	Frm2WcCtrl AT %Q* : UINT;
	{attribute addProperty Name "Frm3Ctrl"}
	Frm3Ctrl AT %Q* : UINT;
	{attribute addProperty Name "Frm3WcCtrl"}
	Frm3WcCtrl AT %Q* : UINT;
	{attribute addProperty Name "Frm4Ctrl"}
	Frm4Ctrl AT %Q* : UINT;
	{attribute addProperty Name "Frm4WcCtrl"}
	Frm4WcCtrl AT %Q* : UINT;
	{attribute addProperty Name "Frm5Ctrl"}
	Frm5Ctrl AT %Q* : UINT;
	{attribute addProperty Name "Frm5WcCtrl"}
	Frm5WcCtrl AT %Q* : UINT;
	{attribute addProperty Name "Frm6Ctrl"}
	Frm6Ctrl AT %Q* : UINT;
	{attribute addProperty Name "Frm6WcCtrl"}
	Frm6WcCtrl AT %Q* : UINT;
	{attribute addProperty Name "Frm7Ctrl"}
	Frm7Ctrl AT %Q* : UINT;
	{attribute addProperty Name "Frm7WcCtrl"}
	Frm7WcCtrl AT %Q* : UINT;
	{attribute addProperty Name "Frm8Ctrl"}
	Frm8Ctrl AT %Q* : UINT;
	{attribute addProperty Name "Frm8WcCtrl"}
	Frm8WcCtrl AT %Q* : UINT;
	{attribute addProperty Name "Frm9Ctrl"}
	Frm9Ctrl AT %Q* : UINT;
	{attribute addProperty Name "Frm9WcCtrl"}
	Frm9WcCtrl AT %Q* : UINT;
	{attribute addProperty Name "Frm10Ctrl"}
	Frm10Ctrl AT %Q* : UINT;
	{attribute addProperty Name "Frm10WcCtrl"}
	Frm10WcCtrl AT %Q* : UINT;
	{attribute addProperty Name "Frm11Ctrl"}
	Frm11Ctrl AT %Q* : UINT;
	{attribute addProperty Name "Frm11WcCtrl"}
	Frm11WcCtrl AT %Q* : UINT;
	{attribute addProperty Name "Frm12Ctrl"}
	Frm12Ctrl AT %Q* : UINT;
	{attribute addProperty Name "Frm12WcCtrl"}
	Frm12WcCtrl AT %Q* : UINT;
	{attribute addProperty Name "Frm13Ctrl"}
	Frm13Ctrl AT %Q* : UINT;
	{attribute addProperty Name "Frm13WcCtrl"}
	Frm13WcCtrl AT %Q* : UINT;
	{attribute addProperty Name "Frm14Ctrl"}
	Frm14Ctrl AT %Q* : UINT;
	{attribute addProperty Name "Frm14WcCtrl"}
	Frm14WcCtrl AT %Q* : UINT;
	{attribute addProperty Name "Frm15Ctrl"}
	Frm15Ctrl AT %Q* : UINT;
	{attribute addProperty Name "Frm15WcCtrl"}
	Frm15WcCtrl AT %Q* : UINT;
	{attribute addProperty Name "Frm16Ctrl"}
	Frm16Ctrl AT %Q* : UINT;
	{attribute addProperty Name "Frm16WcCtrl"}
	Frm16WcCtrl AT %Q* : UINT;
	{attribute addProperty Name "Frm17Ctrl"}
	Frm17Ctrl AT %Q* : UINT;
	{attribute addProperty Name "Frm17WcCtrl"}
	Frm17WcCtrl AT %Q* : UINT;
	{attribute addProperty Name "Frm18Ctrl"}
	Frm18Ctrl AT %Q* : UINT;
	{attribute addProperty Name "Frm18WcCtrl"}
	Frm18WcCtrl AT %Q* : UINT;
	{attribute addProperty Name "Frm19Ctrl"}
	Frm19Ctrl AT %Q* : UINT;
	{attribute addProperty Name "Frm19WcCtrl"}
	Frm19WcCtrl AT %Q* : UINT;
	{attribute addProperty Name "Frm20Ctrl"}
	Frm20Ctrl AT %Q* : UINT;
	{attribute addProperty Name "Frm20WcCtrl"}
	Frm20WcCtrl AT %Q* : UINT;
	{attribute addProperty Name "Frm21Ctrl"}
	Frm21Ctrl AT %Q* : UINT;
	{attribute addProperty Name "Frm21WcCtrl"}
	Frm21WcCtrl AT %Q* : UINT;
	{attribute addProperty Name "Frm22Ctrl"}
	Frm22Ctrl AT %Q* : UINT;
	{attribute addProperty Name "Frm22WcCtrl"}
	Frm22WcCtrl AT %Q* : UINT;
	{attribute addProperty Name "Frm23Ctrl"}
	Frm23Ctrl AT %Q* : UINT;
	{attribute addProperty Name "Frm23WcCtrl"}
	Frm23WcCtrl AT %Q* : UINT;
	{attribute addProperty Name "Frm24Ctrl"}
	Frm24Ctrl AT %Q* : UINT;
	{attribute addProperty Name "Frm24WcCtrl"}
	Frm24WcCtrl AT %Q* : UINT;
	{attribute addProperty Name "Frm25Ctrl"}
	Frm25Ctrl AT %Q* : UINT;
	{attribute addProperty Name "Frm25WcCtrl"}
	Frm25WcCtrl AT %Q* : UINT;
END_STRUCT
END_TYPE

// ---- DUTs/IO/Boxes/EK1100_1FC0878B.TcDUT
{attribute 'GeneratedUsingTerminal: EK1100-0000-0018'}
{attribute addProperty BoxType "EK1100-0000-0018"}
{attribute addProperty Description "EK1100 EtherCAT Coupler (2A E-Bus)"}
{attribute addProperty Physics "YKY"}
{attribute addProperty Id "InfoDataAT %I*InfoData_6F19DB2B2"}
{attribute addProperty CRC "532711307"}
{attribute addProperty Size "2"}
TYPE EK1100_1FC0878B EXTENDS EtcSlaveBoxBase_77A0E4A7 :
STRUCT
	{attribute addProperty Name "InfoData"}
	InfoData : InfoData_6F19DB2B;
END_STRUCT
END_TYPE

// ---- DUTs/IO/Boxes/EK1122_1FC0878B.TcDUT
{attribute 'GeneratedUsingTerminal: EK1122-0000-0018'}
{attribute addProperty BoxType "EK1122-0000-0018"}
{attribute addProperty Description "EK1122 2 port EtherCAT junction"}
{attribute addProperty Physics "KYKY"}
{attribute addProperty Id "InfoDataAT %I*InfoData_6F19DB2B2"}
{attribute addProperty CRC "532711307"}
{attribute addProperty Size "2"}
TYPE EK1122_1FC0878B EXTENDS EtcSlaveTerminalBase_947E5A46 :
STRUCT
	{attribute addProperty Name "InfoData"}
	InfoData : InfoData_6F19DB2B;
END_STRUCT
END_TYPE

// ---- DUTs/IO/Boxes/AT2020_2EA6C9BF.TcDUT
{attribute 'GeneratedUsingTerminal: AT2020-0250-0019'}
{attribute addProperty BoxType "AT2020-0250-0019"}
{attribute addProperty Description "AT2020-0250 Motor module, +22.5°, 250mm, 50V"}
{attribute addProperty Physics "YKY"}
{attribute addProperty Id "CC_InputsAT %I*CC_Inputs_2C1C9EE032CC_OutputsAT %Q*CC_Outputs_69F9BE1432WcStateAT %I*WcState_9091E0EB2InfoDataAT %I*InfoData_BEF6B88E18"}
{attribute addProperty CRC "782682559"}
{attribute addProperty Size "84"}
TYPE AT2020_2EA6C9BF EXTENDS EtcSlaveBoxBase_77A0E4A7 :
STRUCT
	{attribute addProperty Name "CC_Inputs"}
	CC_Inputs : CC_Inputs_2C1C9EE0;
	{attribute addProperty Name "CC_Outputs"}
	CC_Outputs : CC_Outputs_69F9BE14;
	{attribute addProperty Name "WcState"}
	WcState : WcState_9091E0EB;
	{attribute addProperty Name "InfoData"}
	InfoData : InfoData_BEF6B88E;
END_STRUCT
END_TYPE

// ---- DUTs/IO/Boxes/AT2050_33A3DF1B.TcDUT
{attribute 'GeneratedUsingTerminal: AT2050-5500-0018'}
{attribute addProperty BoxType "AT2050-5500-0018"}
{attribute addProperty Description "AT2050-5500 Sensor line 90° clothoid, EtherCAT In"}
{attribute addProperty Physics "K"}
{attribute addProperty Id "FB_InputsAT %I*FB_Inputs_4BC4AA0166FB_OutputsAT %Q*FB_Outputs_DAFD38E02WcStateAT %I*WcState_9091E0EB2InfoDataAT %I*InfoData_A7436BC610"}
{attribute addProperty CRC "866377499"}
{attribute addProperty Size "80"}
TYPE AT2050_33A3DF1B EXTENDS EtcSlaveTerminalBase_947E5A46 :
STRUCT
	{attribute addProperty Name "FB_Inputs"}
	FB_Inputs : FB_Inputs_4BC4AA01;
	{attribute addProperty Name "FB_Outputs"}
	FB_Outputs : FB_Outputs_DAFD38E0;
	{attribute addProperty Name "WcState"}
	WcState : WcState_9091E0EB;
	{attribute addProperty Name "InfoData"}
	InfoData : InfoData_A7436BC6;
END_STRUCT
END_TYPE

// ---- DUTs/IO/Boxes/AT2000_1809CD2F.TcDUT
{attribute 'GeneratedUsingTerminal: AT2000-0233-0022'}
{attribute addProperty BoxType "AT2000-0233-0022"}
{attribute addProperty Description "AT2000-0233 Motor module 233 mm, 48V"}
{attribute addProperty Physics "YKY"}
{attribute addProperty Id "CC_Inputs_14_ChAT %I*CC_Inputs_14_Ch_F1B7955430CC_Outputs_14_ChAT %Q*CC_Outputs_14_Ch_4596551130WcStateAT %I*WcState_9091E0EB2InfoDataAT %I*InfoData_BEF6B88E18"}
{attribute addProperty CRC "403295535"}
{attribute addProperty Size "80"}
TYPE AT2000_1809CD2F EXTENDS EtcSlaveBoxBase_77A0E4A7 :
STRUCT
	{attribute addProperty Name "CC_Inputs_14_Ch"}
	CC_Inputs_14_Ch : CC_Inputs_14_Ch_F1B79554;
	{attribute addProperty Name "CC_Outputs_14_Ch"}
	CC_Outputs_14_Ch : CC_Outputs_14_Ch_45965511;
	{attribute addProperty Name "WcState"}
	WcState : WcState_9091E0EB;
	{attribute addProperty Name "InfoData"}
	InfoData : InfoData_BEF6B88E;
END_STRUCT
END_TYPE

// ---- DUTs/IO/Boxes/AT2000_2EA6C9BF.TcDUT
{attribute 'GeneratedUsingTerminal: AT2000-0250-0016'}
{attribute addProperty BoxType "AT2000-0250-0016"}
{attribute addProperty Description "AT2000-0250 Motor module 250 mm, 50V"}
{attribute addProperty Physics "YKY"}
{attribute addProperty Id "CC_InputsAT %I*CC_Inputs_2C1C9EE032CC_OutputsAT %Q*CC_Outputs_69F9BE1432WcStateAT %I*WcState_9091E0EB2InfoDataAT %I*InfoData_BEF6B88E18"}
{attribute addProperty CRC "782682559"}
{attribute addProperty Size "84"}
TYPE AT2000_2EA6C9BF EXTENDS EtcSlaveBoxBase_77A0E4A7 :
STRUCT
	{attribute addProperty Name "CC_Inputs"}
	CC_Inputs : CC_Inputs_2C1C9EE0;
	{attribute addProperty Name "CC_Outputs"}
	CC_Outputs : CC_Outputs_69F9BE14;
	{attribute addProperty Name "WcState"}
	WcState : WcState_9091E0EB;
	{attribute addProperty Name "InfoData"}
	InfoData : InfoData_BEF6B88E;
END_STRUCT
END_TYPE

// ---- DUTs/IO/Boxes/AT2001_2EA6C9BF.TcDUT
{attribute 'GeneratedUsingTerminal: AT2001-0250-0016'}
{attribute addProperty BoxType "AT2001-0250-0016"}
{attribute addProperty Description "AT2001-0250 Motor module with feed 250 mm, 50V"}
{attribute addProperty Physics "YKY"}
{attribute addProperty Id "CC_InputsAT %I*CC_Inputs_2C1C9EE032CC_OutputsAT %Q*CC_Outputs_69F9BE1432WcStateAT %I*WcState_9091E0EB2InfoDataAT %I*InfoData_BEF6B88E18"}
{attribute addProperty CRC "782682559"}
{attribute addProperty Size "84"}
TYPE AT2001_2EA6C9BF EXTENDS EtcSlaveBoxBase_77A0E4A7 :
STRUCT
	{attribute addProperty Name "CC_Inputs"}
	CC_Inputs : CC_Inputs_2C1C9EE0;
	{attribute addProperty Name "CC_Outputs"}
	CC_Outputs : CC_Outputs_69F9BE14;
	{attribute addProperty Name "WcState"}
	WcState : WcState_9091E0EB;
	{attribute addProperty Name "InfoData"}
	InfoData : InfoData_BEF6B88E;
END_STRUCT
END_TYPE

// ---- DUTs/IO/Boxes/AT2002_2EA6C9BF.TcDUT
{attribute 'GeneratedUsingTerminal: AT2002-0249-0021'}
{attribute addProperty BoxType "AT2002-0249-0021"}
{attribute addProperty Description "AT2002-0249 Motor module (Track management) with feed 249 mm, 48V"}
{attribute addProperty Physics "YKY"}
{attribute addProperty Id "CC_InputsAT %I*CC_Inputs_2C1C9EE032CC_OutputsAT %Q*CC_Outputs_69F9BE1432WcStateAT %I*WcState_9091E0EB2InfoDataAT %I*InfoData_BEF6B88E18"}
{attribute addProperty CRC "782682559"}
{attribute addProperty Size "84"}
TYPE AT2002_2EA6C9BF EXTENDS EtcSlaveBoxBase_77A0E4A7 :
STRUCT
	{attribute addProperty Name "CC_Inputs"}
	CC_Inputs : CC_Inputs_2C1C9EE0;
	{attribute addProperty Name "CC_Outputs"}
	CC_Outputs : CC_Outputs_69F9BE14;
	{attribute addProperty Name "WcState"}
	WcState : WcState_9091E0EB;
	{attribute addProperty Name "InfoData"}
	InfoData : InfoData_BEF6B88E;
END_STRUCT
END_TYPE

// ---- DUTs/IO/Boxes/AT2021_2EA6C9BF.TcDUT
{attribute 'GeneratedUsingTerminal: AT2021-0250-0018'}
{attribute addProperty BoxType "AT2021-0250-0018"}
{attribute addProperty Description "AT2021-0250 Motor module with feed , +22.5°, 250mm, 50V"}
{attribute addProperty Physics "YKY"}
{attribute addProperty Id "CC_InputsAT %I*CC_Inputs_2C1C9EE032CC_OutputsAT %Q*CC_Outputs_69F9BE1432WcStateAT %I*WcState_9091E0EB2InfoDataAT %I*InfoData_BEF6B88E18"}
{attribute addProperty CRC "782682559"}
{attribute addProperty Size "84"}
TYPE AT2021_2EA6C9BF EXTENDS EtcSlaveBoxBase_77A0E4A7 :
STRUCT
	{attribute addProperty Name "CC_Inputs"}
	CC_Inputs : CC_Inputs_2C1C9EE0;
	{attribute addProperty Name "CC_Outputs"}
	CC_Outputs : CC_Outputs_69F9BE14;
	{attribute addProperty Name "WcState"}
	WcState : WcState_9091E0EB;
	{attribute addProperty Name "InfoData"}
	InfoData : InfoData_BEF6B88E;
END_STRUCT
END_TYPE

// ---- DUTs/IO/Boxes/AT2025_2EA6C9BF.TcDUT
{attribute 'GeneratedUsingTerminal: AT2025-0250-0018'}
{attribute addProperty BoxType "AT2025-0250-0018"}
{attribute addProperty Description "AT2025-0250 Motor module, -22.5°, 250mm, 50V"}
{attribute addProperty Physics "YKY"}
{attribute addProperty Id "CC_InputsAT %I*CC_Inputs_2C1C9EE032CC_OutputsAT %Q*CC_Outputs_69F9BE1432WcStateAT %I*WcState_9091E0EB2InfoDataAT %I*InfoData_BEF6B88E18"}
{attribute addProperty CRC "782682559"}
{attribute addProperty Size "84"}
TYPE AT2025_2EA6C9BF EXTENDS EtcSlaveBoxBase_77A0E4A7 :
STRUCT
	{attribute addProperty Name "CC_Inputs"}
	CC_Inputs : CC_Inputs_2C1C9EE0;
	{attribute addProperty Name "CC_Outputs"}
	CC_Outputs : CC_Outputs_69F9BE14;
	{attribute addProperty Name "WcState"}
	WcState : WcState_9091E0EB;
	{attribute addProperty Name "InfoData"}
	InfoData : InfoData_BEF6B88E;
END_STRUCT
END_TYPE

// ---- DUTs/IO/Boxes/AT2026_2EA6C9BF.TcDUT
{attribute 'GeneratedUsingTerminal: AT2026-0250-0021'}
{attribute addProperty BoxType "AT2026-0250-0021"}
{attribute addProperty Description "AT2026-0250 Motor module with feed, -22.5°, 250mm, 48V"}
{attribute addProperty Physics "YKY"}
{attribute addProperty Id "CC_InputsAT %I*CC_Inputs_2C1C9EE032CC_OutputsAT %Q*CC_Outputs_69F9BE1432WcStateAT %I*WcState_9091E0EB2InfoDataAT %I*InfoData_BEF6B88E18"}
{attribute addProperty CRC "782682559"}
{attribute addProperty Size "84"}
TYPE AT2026_2EA6C9BF EXTENDS EtcSlaveBoxBase_77A0E4A7 :
STRUCT
	{attribute addProperty Name "CC_Inputs"}
	CC_Inputs : CC_Inputs_2C1C9EE0;
	{attribute addProperty Name "CC_Outputs"}
	CC_Outputs : CC_Outputs_69F9BE14;
	{attribute addProperty Name "WcState"}
	WcState : WcState_9091E0EB;
	{attribute addProperty Name "InfoData"}
	InfoData : InfoData_BEF6B88E;
END_STRUCT
END_TYPE

// ---- DUTs/IO/Boxes/AT2040_2EA6C9BF.TcDUT
{attribute 'GeneratedUsingTerminal: AT2040-0250-0018'}
{attribute addProperty BoxType "AT2040-0250-0018"}
{attribute addProperty Description "AT2040-0250 Motor module, +45°, 250mm, 50V"}
{attribute addProperty Physics "YKY"}
{attribute addProperty Id "CC_InputsAT %I*CC_Inputs_2C1C9EE032CC_OutputsAT %Q*CC_Outputs_69F9BE1432WcStateAT %I*WcState_9091E0EB2InfoDataAT %I*InfoData_BEF6B88E18"}
{attribute addProperty CRC "782682559"}
{attribute addProperty Size "84"}
TYPE AT2040_2EA6C9BF EXTENDS EtcSlaveBoxBase_77A0E4A7 :
STRUCT
	{attribute addProperty Name "CC_Inputs"}
	CC_Inputs : CC_Inputs_2C1C9EE0;
	{attribute addProperty Name "CC_Outputs"}
	CC_Outputs : CC_Outputs_69F9BE14;
	{attribute addProperty Name "WcState"}
	WcState : WcState_9091E0EB;
	{attribute addProperty Name "InfoData"}
	InfoData : InfoData_BEF6B88E;
END_STRUCT
END_TYPE

// ---- DUTs/IO/Boxes/AT2000_33A3DF1B.TcDUT
{attribute 'GeneratedUsingTerminal: AT2000-5233-0019'}
{attribute addProperty BoxType "AT2000-5233-0019"}
{attribute addProperty Description "AT2000-5233 Sensor line 233 mm"}
{attribute addProperty Physics "K"}
{attribute addProperty Id "FB_InputsAT %I*FB_Inputs_4BC4AA0166FB_OutputsAT %Q*FB_Outputs_DAFD38E02WcStateAT %I*WcState_9091E0EB2InfoDataAT %I*InfoData_A7436BC610"}
{attribute addProperty CRC "866377499"}
{attribute addProperty Size "80"}
TYPE AT2000_33A3DF1B EXTENDS EtcSlaveTerminalBase_947E5A46 :
STRUCT
	{attribute addProperty Name "FB_Inputs"}
	FB_Inputs : FB_Inputs_4BC4AA01;
	{attribute addProperty Name "FB_Outputs"}
	FB_Outputs : FB_Outputs_DAFD38E0;
	{attribute addProperty Name "WcState"}
	WcState : WcState_9091E0EB;
	{attribute addProperty Name "InfoData"}
	InfoData : InfoData_A7436BC6;
END_STRUCT
END_TYPE

// ---- DUTs/IO/Boxes/AT2026_33A3DF1B.TcDUT
{attribute 'GeneratedUsingTerminal: AT2026-5250-0019'}
{attribute addProperty BoxType "AT2026-5250-0019"}
{attribute addProperty Description "AT2026-5250 Sensor line with feed, -22.5°"}
{attribute addProperty Physics "K"}
{attribute addProperty Id "FB_InputsAT %I*FB_Inputs_4BC4AA0166FB_OutputsAT %Q*FB_Outputs_DAFD38E02WcStateAT %I*WcState_9091E0EB2InfoDataAT %I*InfoData_A7436BC610"}
{attribute addProperty CRC "866377499"}
{attribute addProperty Size "80"}
TYPE AT2026_33A3DF1B EXTENDS EtcSlaveTerminalBase_947E5A46 :
STRUCT
	{attribute addProperty Name "FB_Inputs"}
	FB_Inputs : FB_Inputs_4BC4AA01;
	{attribute addProperty Name "FB_Outputs"}
	FB_Outputs : FB_Outputs_DAFD38E0;
	{attribute addProperty Name "WcState"}
	WcState : WcState_9091E0EB;
	{attribute addProperty Name "InfoData"}
	InfoData : InfoData_A7436BC6;
END_STRUCT
END_TYPE

// ---- DUTs/IO/Boxes/AT2041_2EA6C9BF.TcDUT
{attribute 'GeneratedUsingTerminal: AT2041-0250-0018'}
{attribute addProperty BoxType "AT2041-0250-0018"}
{attribute addProperty Description "AT2041-0250 Motor module with feed, +45°, 250mm, 50V"}
{attribute addProperty Physics "YKY"}
{attribute addProperty Id "CC_InputsAT %I*CC_Inputs_2C1C9EE032CC_OutputsAT %Q*CC_Outputs_69F9BE1432WcStateAT %I*WcState_9091E0EB2InfoDataAT %I*InfoData_BEF6B88E18"}
{attribute addProperty CRC "782682559"}
{attribute addProperty Size "84"}
TYPE AT2041_2EA6C9BF EXTENDS EtcSlaveBoxBase_77A0E4A7 :
STRUCT
	{attribute addProperty Name "CC_Inputs"}
	CC_Inputs : CC_Inputs_2C1C9EE0;
	{attribute addProperty Name "CC_Outputs"}
	CC_Outputs : CC_Outputs_69F9BE14;
	{attribute addProperty Name "WcState"}
	WcState : WcState_9091E0EB;
	{attribute addProperty Name "InfoData"}
	InfoData : InfoData_BEF6B88E;
END_STRUCT
END_TYPE

